LIN {X 0,Y 469.098,Z 495.476,A -85,B 0,C 180,E1 -7636.682,E2 -7636.682} C_VEL
LIN {X 0,Y 468.654,Z 505.589,A -85,B 0,C 180,E1 -7637.503,E2 -7637.503} C_VEL
LIN {X 0,Y 468.178,Z 515.821,A -85,B 0,C 180,E1 -7638.527,E2 -7638.527} C_VEL
LIN {X 0,Y 467.646,Z 524.67,A -85,B 0,C 180,E1 -7639.61,E2 -7639.61} C_VEL
LIN {X 0,Y 467.275,Z 533.304,A -85,B 0,C 180,E1 -7640.913,E2 -7640.913} C_VEL
LIN {X 0,Y 467.012,Z 540.205,A -85,B 0,C 180,E1 -7642.216,E2 -7642.216} C_VEL
LIN {X 0,Y 466.802,Z 545.87,A -85,B 0,C 180,E1 -7643.552,E2 -7643.552} C_VEL
LIN {X 0,Y 466.743,Z 550.076,A -85,B 0,C 180,E1 -7644.816,E2 -7644.816} C_VEL
LIN {X 0,Y 466.652,Z 552.371,A -85,B 0,C 180,E1 -7645.681,E2 -7645.681} C_VEL
LIN {X 0,Y 466.691,Z 554.235,A -85,B 0,C 180,E1 -7646.546,E2 -7646.546} C_VEL
LIN {X 0,Y 466.662,Z 555.631,A -85,B 0,C 180,E1 -7647.41,E2 -7647.41} C_VEL
LIN {X 0,Y 466.618,Z 557.235,A -85,B 0,C 180,E1 -7649.137,E2 -7649.137} C_VEL
LIN {X 0,Y 466.598,Z 557.451,A -85,B 0,C 180,E1 -7650,E2 -7650} C_VEL
LIN {X 0,Y 466.618,Z 557.235,A -85,B 0,C 180,E1 -7650.863,E2 -7650.863} C_VEL
LIN {X 0,Y 466.662,Z 555.634,A -85,B 0,C 180,E1 -7652.589,E2 -7652.589} C_VEL
LIN {X 0,Y 466.691,Z 554.239,A -85,B 0,C 180,E1 -7653.453,E2 -7653.453} C_VEL
LIN {X 0,Y 466.694,Z 551.302,A -85,B 0,C 180,E1 -7654.751,E2 -7654.751} C_VEL
LIN {X 0,Y 466.778,Z 547.328,A -85,B 0,C 180,E1 -7656.05,E2 -7656.05} C_VEL
LIN {X 0,Y 466.979,Z 541.219,A -85,B 0,C 180,E1 -7657.567,E2 -7657.567} C_VEL
LIN {X 0,Y 467.24,Z 534.542,A -85,B 0,C 180,E1 -7658.869,E2 -7658.869} C_VEL
LIN {X 0,Y 467.587,Z 526.257,A -85,B 0,C 180,E1 -7660.172,E2 -7660.172} C_VEL
LIN {X 0,Y 468.054,Z 517.77,A -85,B 0,C 180,E1 -7661.256,E2 -7661.256} C_VEL
LIN {X 0,Y 468.531,Z 507.664,A -85,B 0,C 180,E1 -7662.306,E2 -7662.306} C_VEL
LIN {X 0,Y 469.029,Z 495.903,A -85,B 0,C 180,E1 -7663.286,E2 -7663.286} C_VEL
LIN {X 0,Y 469.583,Z 483.606,A -85,B 0,C 180,E1 -7664.076,E2 -7664.076} C_VEL
LIN {X 0,Y 470.068,Z 471.26,A -85,B 0,C 180,E1 -7664.669,E2 -7664.669} C_VEL
LIN {X 0,Y 468.242,Z 458.397,A -85,B 0,C 180,E1 -7665.176,E2 -7665.176} C_VEL
LIN {X 0,Y 466.978,Z 450.681,A -85,B 0,C 180,E1 -7665.416,E2 -7665.416} C_VEL
LIN {X 0,Y 467.142,Z 442.978,A -85,B 0,C 180,E1 -7668.591,E2 -7668.591} C_VEL
LIN {X 0,Y 467.356,Z 435.681,A -85,B 0,C 180,E1 -7671.618,E2 -7671.618} C_VEL
LIN {X 0,Y 467.577,Z 427.867,A -85,B 0,C 180,E1 -7674.889,E2 -7674.889} C_VEL
LIN {X 0,Y 467.867,Z 420.073,A -85,B 0,C 180,E1 -7678.24,E2 -7678.24} C_VEL
LIN {X 0,Y 468.152,Z 413.506,A -85,B 0,C 180,E1 -7681.163,E2 -7681.163} C_VEL
LIN {X 0,Y 468.441,Z 407.928,A -85,B 0,C 180,E1 -7683.718,E2 -7683.718} C_VEL
LIN {X 0,Y 468.502,Z 403.343,A -85,B 0,C 180,E1 -7685.899,E2 -7685.899} C_VEL
LIN {X 0,Y 467.759,Z 397.999,A -85,B 0,C 180,E1 -7688.621,E2 -7688.621} C_VEL
LIN {X 0,Y 467.622,Z 397.24,A -85,B 0,C 180,E1 -7689.141,E2 -7689.141} C_VEL
LIN {X 0,Y 467.588,Z 397.241,A -85,B 0,C 180,E1 -7692.567,E2 -7692.567} C_VEL
LIN {X 0,Y 467.572,Z 397.243,A -85,B 0,C 180,E1 -7695.053,E2 -7695.053} C_VEL
LIN {X 0,Y 467.59,Z 397.24,A -85,B 0,C 180,E1 -7697.44,E2 -7697.44} C_VEL
LIN {X 0,Y 467.584,Z 397.243,A -85,B 0,C 180,E1 -7700.855,E2 -7700.855} C_VEL
LIN {X 0,Y 467.564,Z 397.244,A -85,B 0,C 180,E1 -7704.26,E2 -7704.26} C_VEL
LIN {X 0,Y 467.583,Z 397.243,A -85,B 0,C 180,E1 -7707.321,E2 -7707.321} C_VEL
LIN {X 0,Y 467.572,Z 397.244,A -85,B 0,C 180,E1 -7710.667,E2 -7710.667} C_VEL
LIN {X 0,Y 467.614,Z 397.236,A -85,B 0,C 180,E1 -7713.199,E2 -7713.199} C_VEL
LIN {X 0,Y 467.592,Z 397.241,A -85,B 0,C 180,E1 -7716.469,E2 -7716.469} C_VEL
LIN {X 0,Y 467.626,Z 397.236,A -85,B 0,C 180,E1 -7719.777,E2 -7719.777} C_VEL
LIN {X 0,Y 467.611,Z 397.239,A -85,B 0,C 180,E1 -7722.507,E2 -7722.507} C_VEL
LIN {X 0,Y 467.608,Z 397.235,A -85,B 0,C 180,E1 -7725.197,E2 -7725.197} C_VEL
LIN {X 0,Y 467.685,Z 397.228,A -85,B 0,C 180,E1 -7727.855,E2 -7727.855} C_VEL
LIN {X 0,Y 467.684,Z 397.228,A -85,B 0,C 180,E1 -7731.357,E2 -7731.357} C_VEL
LIN {X 0,Y 467.745,Z 397.22,A -85,B 0,C 180,E1 -7733.963,E2 -7733.963} C_VEL
LIN {X 0,Y 467.861,Z 397.204,A -85,B 0,C 180,E1 -7737.417,E2 -7737.417} C_VEL
LIN {X 0,Y 467.885,Z 397.206,A -85,B 0,C 180,E1 -7740,E2 -7740} C_VEL
LIN {X 0,Y 467.86,Z 397.206,A -85,B 0,C 180,E1 -7742.583,E2 -7742.583} C_VEL
LIN {X 0,Y 467.746,Z 397.221,A -85,B 0,C 180,E1 -7746.037,E2 -7746.037} C_VEL
LIN {X 0,Y 467.684,Z 397.229,A -85,B 0,C 180,E1 -7748.643,E2 -7748.643} C_VEL
LIN {X 0,Y 467.685,Z 397.23,A -85,B 0,C 180,E1 -7752.145,E2 -7752.145} C_VEL
LIN {X 0,Y 467.651,Z 397.233,A -85,B 0,C 180,E1 -7755.885,E2 -7755.885} C_VEL
LIN {X 0,Y 467.625,Z 397.237,A -85,B 0,C 180,E1 -7759.308,E2 -7759.308} C_VEL
LIN {X 0,Y 467.536,Z 397.25,A -85,B 0,C 180,E1 -7762.074,E2 -7762.074} C_VEL
LIN {X 0,Y 467.587,Z 397.238,A -85,B 0,C 180,E1 -7764.888,E2 -7764.888} C_VEL
LIN {X 0,Y 467.629,Z 397.236,A -85,B 0,C 180,E1 -7767.769,E2 -7767.769} C_VEL
LIN {X 0,Y 467.57,Z 397.244,A -85,B 0,C 180,E1 -7771.045,E2 -7771.045} C_VEL
LIN {X 0,Y 467.592,Z 397.24,A -85,B 0,C 180,E1 -7774.243,E2 -7774.243} C_VEL
LIN {X 0,Y 467.553,Z 397.244,A -85,B 0,C 180,E1 -7777.187,E2 -7777.187} C_VEL
LIN {X 0,Y 467.58,Z 397.239,A -85,B 0,C 180,E1 -7780.265,E2 -7780.265} C_VEL
LIN {X 0,Y 467.588,Z 397.239,A -85,B 0,C 180,E1 -7782.567,E2 -7782.567} C_VEL
LIN {X 0,Y 467.573,Z 397.244,A -85,B 0,C 180,E1 -7785.053,E2 -7785.053} C_VEL
LIN {X 0,Y 467.591,Z 397.241,A -85,B 0,C 180,E1 -7787.44,E2 -7787.44} C_VEL
LIN {X 0,Y 467.584,Z 397.24,A -85,B 0,C 180,E1 -7790.855,E2 -7790.855} C_VEL
LIN {X 0,Y 467.475,Z 397.255,A -85,B 0,C 180,E1 -7794.103,E2 -7794.103} C_VEL
LIN {X 0,Y 467.429,Z 397.919,A -85,B 0,C 180,E1 -7795.156,E2 -7795.156} C_VEL
LIN {X 0,Y 467.372,Z 402.107,A -85,B 0,C 180,E1 -7798.244,E2 -7798.244} C_VEL
LIN {X 0,Y 467.244,Z 406.279,A -85,B 0,C 180,E1 -7801.228,E2 -7801.228} C_VEL
LIN {X 0,Y 467.14,Z 410.962,A -85,B 0,C 180,E1 -7804.514,E2 -7804.514} C_VEL
LIN {X 0,Y 467.04,Z 414.543,A -85,B 0,C 180,E1 -7806.968,E2 -7806.968} C_VEL
LIN {X 0,Y 466.898,Z 418.715,A -85,B 0,C 180,E1 -7809.744,E2 -7809.744} C_VEL
LIN {X 0,Y 466.851,Z 422.911,A -85,B 0,C 180,E1 -7812.478,E2 -7812.478} C_VEL
LIN {X 0,Y 466.817,Z 424.912,A -85,B 0,C 180,E1 -7813.735,E2 -7813.735} C_VEL
LIN {X 0,Y 466.734,Z 426.081,A -85,B 0,C 180,E1 -7814.067,E2 -7814.067} C_VEL
LIN {X 0,Y 466.42,Z 428.863,A -85,B 0,C 180,E1 -7814.419,E2 -7814.419} C_VEL
LIN {X 0,Y 465.81,Z 433.444,A -85,B 0,C 180,E1 -7814.735,E2 -7814.735} C_VEL
LIN {X 0,Y 465.219,Z 437.43,A -85,B 0,C 180,E1 -7814.919,E2 -7814.919} C_VEL
LIN {X 0,Y 463.985,Z 445.772,A -85,B 0,C 180,E1 -7815.2,E2 -7815.2} C_VEL
LIN {X 0,Y 463.149,Z 452.928,A -85,B 0,C 180,E1 -7815.511,E2 -7815.511} C_VEL
LIN {X 0,Y 462.676,Z 464.1,A -85,B 0,C 180,E1 -7816.159,E2 -7816.159} C_VEL
LIN {X 0,Y 462.246,Z 474.476,A -85,B 0,C 180,E1 -7816.929,E2 -7816.929} C_VEL
LIN {X 0,Y 461.72,Z 485.163,A -85,B 0,C 180,E1 -7817.919,E2 -7817.919} C_VEL
LIN {X 0,Y 461.147,Z 494.78,A -85,B 0,C 180,E1 -7819.018,E2 -7819.018} C_VEL
LIN {X 0,Y 460.748,Z 502.654,A -85,B 0,C 180,E1 -7820.119,E2 -7820.119} C_VEL
LIN {X 0,Y 460.319,Z 510.353,A -85,B 0,C 180,E1 -7821.439,E2 -7821.439} C_VEL
LIN {X 0,Y 459.943,Z 517.415,A -85,B 0,C 180,E1 -7822.979,E2 -7822.979} C_VEL
LIN {X 0,Y 459.872,Z 522.116,A -85,B 0,C 180,E1 -7824.299,E2 -7824.299} C_VEL
LIN {X 0,Y 459.676,Z 525.72,A -85,B 0,C 180,E1 -7825.616,E2 -7825.616} C_VEL
LIN {X 0,Y 459.707,Z 527.58,A -85,B 0,C 180,E1 -7826.494,E2 -7826.494} C_VEL
LIN {X 0,Y 459.608,Z 528.985,A -85,B 0,C 180,E1 -7827.371,E2 -7827.371} C_VEL
LIN {X 0,Y 459.523,Z 530.598,A -85,B 0,C 180,E1 -7829.124,E2 -7829.124} C_VEL
LIN {X 0,Y 459.53,Z 530.833,A -85,B 0,C 180,E1 -7830,E2 -7830} C_VEL
LIN {X 0,Y 459.523,Z 530.646,A -85,B 0,C 180,E1 -7830.876,E2 -7830.876} C_VEL
LIN {X 0,Y 459.608,Z 529.096,A -85,B 0,C 180,E1 -7832.629,E2 -7832.629} C_VEL
LIN {X 0,Y 459.689,Z 527.741,A -85,B 0,C 180,E1 -7833.506,E2 -7833.506} C_VEL
LIN {X 0,Y 459.671,Z 524.88,A -85,B 0,C 180,E1 -7834.824,E2 -7834.824} C_VEL
LIN {X 0,Y 459.921,Z 520.994,A -85,B 0,C 180,E1 -7836.141,E2 -7836.141} C_VEL
LIN {X 0,Y 460.047,Z 515.986,A -85,B 0,C 180,E1 -7837.461,E2 -7837.461} C_VEL
LIN {X 0,Y 460.375,Z 509.678,A -85,B 0,C 180,E1 -7838.781,E2 -7838.781} C_VEL
LIN {X 0,Y 460.73,Z 501.782,A -85,B 0,C 180,E1 -7840.103,E2 -7840.103} C_VEL
LIN {X 0,Y 461.286,Z 491.956,A -85,B 0,C 180,E1 -7841.424,E2 -7841.424} C_VEL
LIN {X 0,Y 461.937,Z 481.725,A -85,B 0,C 180,E1 -7842.514,E2 -7842.514} C_VEL
LIN {X 0,Y 462.338,Z 470.839,A -85,B 0,C 180,E1 -7843.451,E2 -7843.451} C_VEL
LIN {X 0,Y 462.833,Z 460.258,A -85,B 0,C 180,E1 -7844.173,E2 -7844.173} C_VEL
LIN {X 0,Y 463.274,Z 447.688,A -85,B 0,C 180,E1 -7844.833,E2 -7844.833} C_VEL
LIN {X 0,Y 463.206,Z 443.667,A -85,B 0,C 180,E1 -7845.01,E2 -7845.01} C_VEL
LIN {X 0,Y 460.798,Z 431.07,A -85,B 0,C 180,E1 -7845.515,E2 -7845.515} C_VEL
LIN {X 0,Y 459.769,Z 426.584,A -85,B 0,C 180,E1 -7845.672,E2 -7845.672} C_VEL
LIN {X 0,Y 459.841,Z 421.829,A -85,B 0,C 180,E1 -7848.721,E2 -7848.721} C_VEL
LIN {X 0,Y 459.92,Z 416.213,A -85,B 0,C 180,E1 -7852.459,E2 -7852.459} C_VEL
LIN {X 0,Y 460.066,Z 411.592,A -85,B 0,C 180,E1 -7855.672,E2 -7855.672} C_VEL
LIN {X 0,Y 460.258,Z 406.541,A -85,B 0,C 180,E1 -7859.251,E2 -7859.251} C_VEL
LIN {X 0,Y 460.328,Z 402.349,A -85,B 0,C 180,E1 -7862.301,E2 -7862.301} C_VEL
LIN {X 0,Y 460.414,Z 399.416,A -85,B 0,C 180,E1 -7864.484,E2 -7864.484} C_VEL
LIN {X 0,Y 460.367,Z 398.143,A -85,B 0,C 180,E1 -7865.459,E2 -7865.459} C_VEL
LIN {X 0,Y 460.499,Z 398.121,A -85,B 0,C 180,E1 -7867.624,E2 -7867.624} C_VEL
LIN {X 0,Y 460.546,Z 398.118,A -85,B 0,C 180,E1 -7870.27,E2 -7870.27} C_VEL
LIN {X 0,Y 460.511,Z 398.123,A -85,B 0,C 180,E1 -7873.374,E2 -7873.374} C_VEL
LIN {X 0,Y 460.499,Z 398.124,A -85,B 0,C 180,E1 -7876.624,E2 -7876.624} C_VEL
LIN {X 0,Y 460.545,Z 398.115,A -85,B 0,C 180,E1 -7879.731,E2 -7879.731} C_VEL
LIN {X 0,Y 460.529,Z 398.122,A -85,B 0,C 180,E1 -7882.52,E2 -7882.52} C_VEL
LIN {X 0,Y 460.549,Z 398.117,A -85,B 0,C 180,E1 -7885.624,E2 -7885.624} C_VEL
LIN {X 0,Y 460.54,Z 398.12,A -85,B 0,C 180,E1 -7888.745,E2 -7888.745} C_VEL
LIN {X 0,Y 460.592,Z 398.113,A -85,B 0,C 180,E1 -7892.252,E2 -7892.252} C_VEL
LIN {X 0,Y 460.534,Z 398.117,A -85,B 0,C 180,E1 -7895.667,E2 -7895.667} C_VEL
LIN {X 0,Y 460.524,Z 398.12,A -85,B 0,C 180,E1 -7898.578,E2 -7898.578} C_VEL
LIN {X 0,Y 460.59,Z 398.112,A -85,B 0,C 180,E1 -7901.311,E2 -7901.311} C_VEL
LIN {X 0,Y 460.607,Z 398.11,A -85,B 0,C 180,E1 -7904.059,E2 -7904.059} C_VEL
LIN {X 0,Y 460.613,Z 398.108,A -85,B 0,C 180,E1 -7907.666,E2 -7907.666} C_VEL
LIN {X 0,Y 460.632,Z 398.106,A -85,B 0,C 180,E1 -7911.224,E2 -7911.224} C_VEL
LIN {X 0,Y 460.713,Z 398.097,A -85,B 0,C 180,E1 -7913.87,E2 -7913.87} C_VEL
LIN {X 0,Y 460.802,Z 398.085,A -85,B 0,C 180,E1 -7917.377,E2 -7917.377} C_VEL
LIN {X 0,Y 460.856,Z 398.082,A -85,B 0,C 180,E1 -7920,E2 -7920} C_VEL
LIN {X 0,Y 460.803,Z 398.083,A -85,B 0,C 180,E1 -7922.622,E2 -7922.622} C_VEL
LIN {X 0,Y 460.713,Z 398.097,A -85,B 0,C 180,E1 -7926.13,E2 -7926.13} C_VEL
LIN {X 0,Y 460.632,Z 398.107,A -85,B 0,C 180,E1 -7928.776,E2 -7928.776} C_VEL
LIN {X 0,Y 460.638,Z 398.105,A -85,B 0,C 180,E1 -7932.457,E2 -7932.457} C_VEL
LIN {X 0,Y 460.603,Z 398.109,A -85,B 0,C 180,E1 -7935.997,E2 -7935.997} C_VEL
LIN {X 0,Y 460.575,Z 398.115,A -85,B 0,C 180,E1 -7938.902,E2 -7938.902} C_VEL
LIN {X 0,Y 460.519,Z 398.121,A -85,B 0,C 180,E1 -7941.486,E2 -7941.486} C_VEL
LIN {X 0,Y 460.534,Z 398.118,A -85,B 0,C 180,E1 -7944.333,E2 -7944.333} C_VEL
LIN {X 0,Y 460.591,Z 398.111,A -85,B 0,C 180,E1 -7947.748,E2 -7947.748} C_VEL
LIN {X 0,Y 460.523,Z 398.121,A -85,B 0,C 180,E1 -7951.283,E2 -7951.283} C_VEL
LIN {X 0,Y 460.536,Z 398.12,A -85,B 0,C 180,E1 -7954.506,E2 -7954.506} C_VEL
LIN {X 0,Y 460.531,Z 398.12,A -85,B 0,C 180,E1 -7957.62,E2 -7957.62} C_VEL
LIN {X 0,Y 460.544,Z 398.116,A -85,B 0,C 180,E1 -7960.269,E2 -7960.269} C_VEL
LIN {X 0,Y 460.503,Z 398.122,A -85,B 0,C 180,E1 -7963.375,E2 -7963.375} C_VEL
LIN {X 0,Y 460.512,Z 398.124,A -85,B 0,C 180,E1 -7966.626,E2 -7966.626} C_VEL
LIN {X 0,Y 460.545,Z 398.123,A -85,B 0,C 180,E1 -7969.73,E2 -7969.73} C_VEL
LIN {X 0,Y 460.596,Z 398.172,A -85,B 0,C 180,E1 -7970.781,E2 -7970.781} C_VEL
LIN {X 0,Y 461.478,Z 403.993,A -85,B 0,C 180,E1 -7973.819,E2 -7973.819} C_VEL
LIN {X 0,Y 461.428,Z 408.951,A -85,B 0,C 180,E1 -7976.225,E2 -7976.225} C_VEL
LIN {X 0,Y 461.086,Z 416.657,A -85,B 0,C 180,E1 -7979.801,E2 -7979.801} C_VEL
LIN {X 0,Y 460.697,Z 423.307,A -85,B 0,C 180,E1 -7982.764,E2 -7982.764} C_VEL
LIN {X 0,Y 460.487,Z 429.977,A -85,B 0,C 180,E1 -7985.664,E2 -7985.664} C_VEL
LIN {X 0,Y 460.278,Z 436.992,A -85,B 0,C 180,E1 -7988.656,E2 -7988.656} C_VEL
LIN {X 0,Y 460.04,Z 444.334,A -85,B 0,C 180,E1 -7991.749,E2 -7991.749} C_VEL
LIN {X 0,Y 459.912,Z 450.511,A -85,B 0,C 180,E1 -7994.351,E2 -7994.351} C_VEL
LIN {X 0,Y 462.129,Z 464.356,A -85,B 0,C 180,E1 -7994.812,E2 -7994.812} C_VEL
LIN {X 0,Y 463.103,Z 472.383,A -85,B 0,C 180,E1 -7995.162,E2 -7995.162} C_VEL
LIN {X 0,Y 462.697,Z 483.416,A -85,B 0,C 180,E1 -7995.71,E2 -7995.71} C_VEL
LIN {X 0,Y 462.168,Z 495.274,A -85,B 0,C 180,E1 -7996.479,E2 -7996.479} C_VEL
LIN {X 0,Y 461.66,Z 505.773,A -85,B 0,C 180,E1 -7997.347,E2 -7997.347} C_VEL
LIN {X 0,Y 461.19,Z 515.618,A -85,B 0,C 180,E1 -7998.351,E2 -7998.351} C_VEL
LIN {X 0,Y 460.632,Z 524.467,A -85,B 0,C 180,E1 -7999.45,E2 -7999.45} C_VEL
LIN {X 0,Y 460.241,Z 533.1,A -85,B 0,C 180,E1 -8000.773,E2 -8000.773} C_VEL
LIN {X 0,Y 459.951,Z 540.001,A -85,B 0,C 180,E1 -8002.096,E2 -8002.096} C_VEL
LIN {X 0,Y 459.713,Z 546.099,A -85,B 0,C 180,E1 -8003.57,E2 -8003.57} C_VEL
LIN {X 0,Y 459.622,Z 551.097,A -85,B 0,C 180,E1 -8005.176,E2 -8005.176} C_VEL
LIN {X 0,Y 459.586,Z 554.031,A -85,B 0,C 180,E1 -8006.493,E2 -8006.493} C_VEL
LIN {X 0,Y 459.584,Z 555.428,A -85,B 0,C 180,E1 -8007.37,E2 -8007.37} C_VEL
LIN {X 0,Y 459.521,Z 557.031,A -85,B 0,C 180,E1 -8009.124,E2 -8009.124} C_VEL
LIN {X 0,Y 459.53,Z 557.248,A -85,B 0,C 180,E1 -8010,E2 -8010} C_VEL
LIN {X 0,Y 459.521,Z 557.031,A -85,B 0,C 180,E1 -8010.876,E2 -8010.876} C_VEL
LIN {X 0,Y 459.584,Z 555.43,A -85,B 0,C 180,E1 -8012.629,E2 -8012.629} C_VEL
LIN {X 0,Y 459.586,Z 554.034,A -85,B 0,C 180,E1 -8013.507,E2 -8013.507} C_VEL
LIN {X 0,Y 459.622,Z 551.098,A -85,B 0,C 180,E1 -8014.824,E2 -8014.824} C_VEL
LIN {X 0,Y 459.713,Z 546.096,A -85,B 0,C 180,E1 -8016.43,E2 -8016.43} C_VEL
LIN {X 0,Y 459.951,Z 540,A -85,B 0,C 180,E1 -8017.904,E2 -8017.904} C_VEL
LIN {X 0,Y 460.241,Z 533.098,A -85,B 0,C 180,E1 -8019.226,E2 -8019.226} C_VEL
LIN {X 0,Y 460.632,Z 524.463,A -85,B 0,C 180,E1 -8020.55,E2 -8020.55} C_VEL
LIN {X 0,Y 461.186,Z 515.612,A -85,B 0,C 180,E1 -8021.649,E2 -8021.649} C_VEL
LIN {X 0,Y 461.707,Z 505.837,A -85,B 0,C 180,E1 -8022.645,E2 -8022.645} C_VEL
LIN {X 0,Y 462.142,Z 495.266,A -85,B 0,C 180,E1 -8023.522,E2 -8023.522} C_VEL
LIN {X 0,Y 462.684,Z 483.397,A -85,B 0,C 180,E1 -8024.29,E2 -8024.29} C_VEL
LIN {X 0,Y 463.112,Z 471.048,A -85,B 0,C 180,E1 -8024.894,E2 -8024.894} C_VEL
LIN {X 0,Y 461.147,Z 457.996,A -85,B 0,C 180,E1 -8025.421,E2 -8025.421} C_VEL
LIN {X 0,Y 459.913,Z 450.507,A -85,B 0,C 180,E1 -8025.649,E2 -8025.649} C_VEL
LIN {X 0,Y 460.102,Z 442.235,A -85,B 0,C 180,E1 -8029.126,E2 -8029.126} C_VEL
LIN {X 0,Y 460.306,Z 435.521,A -85,B 0,C 180,E1 -8031.967,E2 -8031.967} C_VEL
LIN {X 0,Y 460.573,Z 427.726,A -85,B 0,C 180,E1 -8035.294,E2 -8035.294} C_VEL
LIN {X 0,Y 460.903,Z 419.951,A -85,B 0,C 180,E1 -8038.706,E2 -8038.706} C_VEL
LIN {X 0,Y 461.171,Z 413.989,A -85,B 0,C 180,E1 -8041.415,E2 -8041.415} C_VEL
LIN {X 0,Y 461.515,Z 407.028,A -85,B 0,C 180,E1 -8044.682,E2 -8044.682} C_VEL
LIN {X 0,Y 461.253,Z 402.369,A -85,B 0,C 180,E1 -8047.003,E2 -8047.003} C_VEL
LIN {X 0,Y 460.56,Z 398.119,A -85,B 0,C 180,E1 -8049.348,E2 -8049.348} C_VEL
LIN {X 0,Y 460.525,Z 398.124,A -85,B 0,C 180,E1 -8052.181,E2 -8052.181} C_VEL
LIN {X 0,Y 460.519,Z 398.124,A -85,B 0,C 180,E1 -8055.411,E2 -8055.411} C_VEL
LIN {X 0,Y 460.533,Z 398.117,A -85,B 0,C 180,E1 -8058.397,E2 -8058.397} C_VEL
LIN {X 0,Y 460.528,Z 398.119,A -85,B 0,C 180,E1 -8061.267,E2 -8061.267} C_VEL
LIN {X 0,Y 460.515,Z 398.123,A -85,B 0,C 180,E1 -8064.555,E2 -8064.555} C_VEL
LIN {X 0,Y 460.533,Z 398.118,A -85,B 0,C 180,E1 -8067.716,E2 -8067.716} C_VEL
LIN {X 0,Y 460.542,Z 398.121,A -85,B 0,C 180,E1 -8070.769,E2 -8070.769} C_VEL
LIN {X 0,Y 460.557,Z 398.114,A -85,B 0,C 180,E1 -8073.734,E2 -8073.734} C_VEL
LIN {X 0,Y 460.546,Z 398.118,A -85,B 0,C 180,E1 -8076.624,E2 -8076.624} C_VEL
LIN {X 0,Y 460.554,Z 398.116,A -85,B 0,C 180,E1 -8079.453,E2 -8079.453} C_VEL
LIN {X 0,Y 460.561,Z 398.115,A -85,B 0,C 180,E1 -8082.23,E2 -8082.23} C_VEL
LIN {X 0,Y 460.567,Z 398.114,A -85,B 0,C 180,E1 -8084.965,E2 -8084.965} C_VEL
LIN {X 0,Y 460.632,Z 398.106,A -85,B 0,C 180,E1 -8087.666,E2 -8087.666} C_VEL
LIN {X 0,Y 460.631,Z 398.107,A -85,B 0,C 180,E1 -8091.224,E2 -8091.224} C_VEL
LIN {X 0,Y 460.712,Z 398.097,A -85,B 0,C 180,E1 -8093.87,E2 -8093.87} C_VEL
LIN {X 0,Y 460.802,Z 398.083,A -85,B 0,C 180,E1 -8097.378,E2 -8097.378} C_VEL
LIN {X 0,Y 460.856,Z 398.081,A -85,B 0,C 180,E1 -8100,E2 -8100} C_VEL
LIN {X 0,Y 460.801,Z 398.085,A -85,B 0,C 180,E1 -8102.623,E2 -8102.623} C_VEL
LIN {X 0,Y 460.712,Z 398.097,A -85,B 0,C 180,E1 -8106.13,E2 -8106.13} C_VEL
LIN {X 0,Y 460.631,Z 398.106,A -85,B 0,C 180,E1 -8108.776,E2 -8108.776} C_VEL
LIN {X 0,Y 460.636,Z 398.105,A -85,B 0,C 180,E1 -8112.457,E2 -8112.457} C_VEL
LIN {X 0,Y 460.602,Z 398.111,A -85,B 0,C 180,E1 -8115.998,E2 -8115.998} C_VEL
LIN {X 0,Y 460.571,Z 398.115,A -85,B 0,C 180,E1 -8119.616,E2 -8119.616} C_VEL
LIN {X 0,Y 460.513,Z 398.121,A -85,B 0,C 180,E1 -8122.429,E2 -8122.429} C_VEL
LIN {X 0,Y 460.555,Z 398.119,A -85,B 0,C 180,E1 -8125.798,E2 -8125.798} C_VEL
LIN {X 0,Y 460.557,Z 398.115,A -85,B 0,C 180,E1 -8128.233,E2 -8128.233} C_VEL
LIN {X 0,Y 460.523,Z 398.122,A -85,B 0,C 180,E1 -8131.283,E2 -8131.283} C_VEL
LIN {X 0,Y 460.536,Z 398.118,A -85,B 0,C 180,E1 -8134.506,E2 -8134.506} C_VEL
LIN {X 0,Y 460.531,Z 398.123,A -85,B 0,C 180,E1 -8137.621,E2 -8137.621} C_VEL
LIN {X 0,Y 460.544,Z 398.115,A -85,B 0,C 180,E1 -8140.27,E2 -8140.27} C_VEL
LIN {X 0,Y 460.502,Z 398.124,A -85,B 0,C 180,E1 -8143.375,E2 -8143.375} C_VEL
LIN {X 0,Y 460.511,Z 398.122,A -85,B 0,C 180,E1 -8146.626,E2 -8146.626} C_VEL
LIN {X 0,Y 460.545,Z 398.118,A -85,B 0,C 180,E1 -8149.731,E2 -8149.731} C_VEL
LIN {X 0,Y 460.495,Z 398.121,A -85,B 0,C 180,E1 -8152.525,E2 -8152.525} C_VEL
LIN {X 0,Y 460.375,Z 398.142,A -85,B 0,C 180,E1 -8154.542,E2 -8154.542} C_VEL
LIN {X 0,Y 460.355,Z 401.412,A -85,B 0,C 180,E1 -8157.104,E2 -8157.104} C_VEL
LIN {X 0,Y 460.26,Z 405.006,A -85,B 0,C 180,E1 -8159.742,E2 -8159.742} C_VEL
LIN {X 0,Y 460.113,Z 409.176,A -85,B 0,C 180,E1 -8162.727,E2 -8162.727} C_VEL
LIN {X 0,Y 460.003,Z 413.321,A -85,B 0,C 180,E1 -8165.637,E2 -8165.637} C_VEL
LIN {X 0,Y 459.851,Z 417.941,A -85,B 0,C 180,E1 -8168.793,E2 -8168.793} C_VEL
LIN {X 0,Y 459.844,Z 421.815,A -85,B 0,C 180,E1 -8171.366,E2 -8171.366} C_VEL
LIN {X 0,Y 459.814,Z 426.595,A -85,B 0,C 180,E1 -8174.429,E2 -8174.429} C_VEL
LIN {X 0,Y 462.668,Z 440.317,A -85,B 0,C 180,E1 -8174.936,E2 -8174.936} C_VEL
LIN {X 0,Y 463.317,Z 445.574,A -85,B 0,C 180,E1 -8175.169,E2 -8175.169} C_VEL
LIN {X 0,Y 463.149,Z 452.928,A -85,B 0,C 180,E1 -8175.511,E2 -8175.511} C_VEL
LIN {X 0,Y 462.255,Z 458.367,A -85,B 0,C 180,E1 -8175.777,E2 -8175.777} C_VEL
LIN {X 0,Y 459.141,Z 467.025,A -85,B 0,C 180,E1 -8176.238,E2 -8176.238} C_VEL
LIN {X 0,Y 456.005,Z 475.282,A -85,B 0,C 180,E1 -8176.795,E2 -8176.795} C_VEL
LIN {X 0,Y 455.08,Z 480.086,A -85,B 0,C 180,E1 -8177.208,E2 -8177.208} C_VEL
LIN {X 0,Y 454.511,Z 489.458,A -85,B 0,C 180,E1 -8178.177,E2 -8178.177} C_VEL
LIN {X 0,Y 454.035,Z 498.302,A -85,B 0,C 180,E1 -8179.295,E2 -8179.295} C_VEL
LIN {X 0,Y 453.531,Z 506.932,A -85,B 0,C 180,E1 -8180.636,E2 -8180.636} C_VEL
LIN {X 0,Y 453.095,Z 513.811,A -85,B 0,C 180,E1 -8181.975,E2 -8181.975} C_VEL
LIN {X 0,Y 452.869,Z 519.329,A -85,B 0,C 180,E1 -8183.32,E2 -8183.32} C_VEL
LIN {X 0,Y 452.695,Z 523.638,A -85,B 0,C 180,E1 -8184.655,E2 -8184.655} C_VEL
LIN {X 0,Y 452.585,Z 525.926,A -85,B 0,C 180,E1 -8185.547,E2 -8185.547} C_VEL
LIN {X 0,Y 452.622,Z 527.785,A -85,B 0,C 180,E1 -8186.439,E2 -8186.439} C_VEL
LIN {X 0,Y 452.535,Z 529.189,A -85,B 0,C 180,E1 -8187.33,E2 -8187.33} C_VEL
LIN {X 0,Y 452.43,Z 530.802,A -85,B 0,C 180,E1 -8189.11,E2 -8189.11} C_VEL
LIN {X 0,Y 452.435,Z 531.037,A -85,B 0,C 180,E1 -8190,E2 -8190} C_VEL
LIN {X 0,Y 452.43,Z 530.85,A -85,B 0,C 180,E1 -8190.89,E2 -8190.89} C_VEL
LIN {X 0,Y 452.534,Z 529.299,A -85,B 0,C 180,E1 -8192.671,E2 -8192.671} C_VEL
LIN {X 0,Y 452.606,Z 527.944,A -85,B 0,C 180,E1 -8193.561,E2 -8193.561} C_VEL
LIN {X 0,Y 452.603,Z 525.083,A -85,B 0,C 180,E1 -8194.899,E2 -8194.899} C_VEL
LIN {X 0,Y 452.85,Z 521.197,A -85,B 0,C 180,E1 -8196.237,E2 -8196.237} C_VEL
LIN {X 0,Y 452.99,Z 516.188,A -85,B 0,C 180,E1 -8197.578,E2 -8197.578} C_VEL
LIN {X 0,Y 453.357,Z 509.88,A -85,B 0,C 180,E1 -8198.918,E2 -8198.918} C_VEL
LIN {X 0,Y 453.743,Z 501.983,A -85,B 0,C 180,E1 -8200.261,E2 -8200.261} C_VEL
LIN {X 0,Y 454.336,Z 492.156,A -85,B 0,C 180,E1 -8201.601,E2 -8201.601} C_VEL
LIN {X 0,Y 455.009,Z 482.059,A -85,B 0,C 180,E1 -8202.694,E2 -8202.694} C_VEL
LIN {X 0,Y 455.414,Z 471.637,A -85,B 0,C 180,E1 -8203.611,E2 -8203.611} C_VEL
LIN {X 0,Y 455.968,Z 460.454,A -85,B 0,C 180,E1 -8204.391,E2 -8204.391} C_VEL
LIN {X 0,Y 456.413,Z 447.882,A -85,B 0,C 180,E1 -8205.061,E2 -8205.061} C_VEL
LIN {X 0,Y 456.031,Z 442.556,A -85,B 0,C 180,E1 -8205.304,E2 -8205.304} C_VEL
LIN {X 0,Y 453.255,Z 429.318,A -85,B 0,C 180,E1 -8205.83,E2 -8205.83} C_VEL
LIN {X 0,Y 452.664,Z 426.786,A -85,B 0,C 180,E1 -8205.922,E2 -8205.922} C_VEL
LIN {X 0,Y 452.774,Z 422.006,A -85,B 0,C 180,E1 -8209.024,E2 -8209.024} C_VEL
LIN {X 0,Y 452.816,Z 417.78,A -85,B 0,C 180,E1 -8211.87,E2 -8211.87} C_VEL
LIN {X 0,Y 452.962,Z 413.615,A -85,B 0,C 180,E1 -8214.767,E2 -8214.767} C_VEL
LIN {X 0,Y 453.077,Z 409.294,A -85,B 0,C 180,E1 -8217.85,E2 -8217.85} C_VEL
LIN {X 0,Y 453.247,Z 405.268,A -85,B 0,C 180,E1 -8220.777,E2 -8220.777} C_VEL
LIN {X 0,Y 453.346,Z 401.055,A -85,B 0,C 180,E1 -8223.924,E2 -8223.924} C_VEL
LIN {X 0,Y 453.353,Z 399.651,A -85,B 0,C 180,E1 -8225.001,E2 -8225.001} C_VEL
LIN {X 0,Y 453.4,Z 399.009,A -85,B 0,C 180,E1 -8226.289,E2 -8226.289} C_VEL
LIN {X 0,Y 453.492,Z 398.995,A -85,B 0,C 180,E1 -8229.45,E2 -8229.45} C_VEL
LIN {X 0,Y 453.481,Z 398.997,A -85,B 0,C 180,E1 -8231.935,E2 -8231.935} C_VEL
LIN {X 0,Y 453.486,Z 398.997,A -85,B 0,C 180,E1 -8235.471,E2 -8235.471} C_VEL
LIN {X 0,Y 453.482,Z 398.997,A -85,B 0,C 180,E1 -8238.209,E2 -8238.209} C_VEL
LIN {X 0,Y 453.513,Z 398.995,A -85,B 0,C 180,E1 -8240.791,E2 -8240.791} C_VEL
LIN {X 0,Y 453.457,Z 399,A -85,B 0,C 180,E1 -8243.917,E2 -8243.917} C_VEL
LIN {X 0,Y 453.486,Z 398.997,A -85,B 0,C 180,E1 -8247.151,E2 -8247.151} C_VEL
LIN {X 0,Y 453.478,Z 398.998,A -85,B 0,C 180,E1 -8250.268,E2 -8250.268} C_VEL
LIN {X 0,Y 453.508,Z 398.991,A -85,B 0,C 180,E1 -8253.294,E2 -8253.294} C_VEL
LIN {X 0,Y 453.501,Z 398.998,A -85,B 0,C 180,E1 -8256.239,E2 -8256.239} C_VEL
LIN {X 0,Y 453.486,Z 398.996,A -85,B 0,C 180,E1 -8259.118,E2 -8259.118} C_VEL
LIN {X 0,Y 453.507,Z 398.995,A -85,B 0,C 180,E1 -8261.944,E2 -8261.944} C_VEL
LIN {X 0,Y 453.543,Z 398.99,A -85,B 0,C 180,E1 -8264.726,E2 -8264.726} C_VEL
LIN {X 0,Y 453.563,Z 398.987,A -85,B 0,C 180,E1 -8268.379,E2 -8268.379} C_VEL
LIN {X 0,Y 453.656,Z 398.977,A -85,B 0,C 180,E1 -8271.985,E2 -8271.985} C_VEL
LIN {X 0,Y 453.673,Z 398.974,A -85,B 0,C 180,E1 -8274.667,E2 -8274.667} C_VEL
LIN {X 0,Y 453.746,Z 398.964,A -85,B 0,C 180,E1 -8277.337,E2 -8277.337} C_VEL
LIN {X 0,Y 453.826,Z 398.957,A -85,B 0,C 180,E1 -8280,E2 -8280} C_VEL
LIN {X 0,Y 453.747,Z 398.962,A -85,B 0,C 180,E1 -8282.663,E2 -8282.663} C_VEL
LIN {X 0,Y 453.68,Z 398.973,A -85,B 0,C 180,E1 -8286.225,E2 -8286.225} C_VEL
LIN {X 0,Y 453.596,Z 398.983,A -85,B 0,C 180,E1 -8288.913,E2 -8288.913} C_VEL
LIN {X 0,Y 453.605,Z 398.98,A -85,B 0,C 180,E1 -8292.551,E2 -8292.551} C_VEL
LIN {X 0,Y 453.548,Z 398.987,A -85,B 0,C 180,E1 -8296.196,E2 -8296.196} C_VEL
LIN {X 0,Y 453.524,Z 398.994,A -85,B 0,C 180,E1 -8299.041,E2 -8299.041} C_VEL
LIN {X 0,Y 453.479,Z 399,A -85,B 0,C 180,E1 -8301.836,E2 -8301.836} C_VEL
LIN {X 0,Y 453.504,Z 398.995,A -85,B 0,C 180,E1 -8304.735,E2 -8304.735} C_VEL
LIN {X 0,Y 453.54,Z 398.988,A -85,B 0,C 180,E1 -8307.961,E2 -8307.961} C_VEL
LIN {X 0,Y 453.468,Z 398.999,A -85,B 0,C 180,E1 -8311.525,E2 -8311.525} C_VEL
LIN {X 0,Y 453.491,Z 398.998,A -85,B 0,C 180,E1 -8314.778,E2 -8314.778} C_VEL
LIN {X 0,Y 453.476,Z 398.998,A -85,B 0,C 180,E1 -8318.311,E2 -8318.311} C_VEL
LIN {X 0,Y 453.496,Z 398.995,A -85,B 0,C 180,E1 -8320.609,E2 -8320.609} C_VEL
LIN {X 0,Y 453.459,Z 399,A -85,B 0,C 180,E1 -8323.244,E2 -8323.244} C_VEL
LIN {X 0,Y 453.476,Z 398.998,A -85,B 0,C 180,E1 -8325.78,E2 -8325.78} C_VEL
LIN {X 0,Y 453.484,Z 399.003,A -85,B 0,C 180,E1 -8328.21,E2 -8328.21} C_VEL
LIN {X 0,Y 453.533,Z 399.042,A -85,B 0,C 180,E1 -8330.555,E2 -8330.555} C_VEL
LIN {X 0,Y 454.425,Z 404.644,A -85,B 0,C 180,E1 -8333.535,E2 -8333.535} C_VEL
LIN {X 0,Y 454.472,Z 408.858,A -85,B 0,C 180,E1 -8335.636,E2 -8335.636} C_VEL
LIN {X 0,Y 454.114,Z 415.52,A -85,B 0,C 180,E1 -8338.807,E2 -8338.807} C_VEL
LIN {X 0,Y 453.881,Z 420.959,A -85,B 0,C 180,E1 -8341.314,E2 -8341.314} C_VEL
LIN {X 0,Y 453.507,Z 428.719,A -85,B 0,C 180,E1 -8344.775,E2 -8344.775} C_VEL
LIN {X 0,Y 453.237,Z 436.47,A -85,B 0,C 180,E1 -8348.152,E2 -8348.152} C_VEL
LIN {X 0,Y 453.005,Z 443.441,A -85,B 0,C 180,E1 -8351.15,E2 -8351.15} C_VEL
LIN {X 0,Y 452.869,Z 450.487,A -85,B 0,C 180,E1 -8354.112,E2 -8354.112} C_VEL
LIN {X 0,Y 455.035,Z 463.693,A -85,B 0,C 180,E1 -8354.552,E2 -8354.552} C_VEL
LIN {X 0,Y 456.209,Z 473.487,A -85,B 0,C 180,E1 -8354.989,E2 -8354.989} C_VEL
LIN {X 0,Y 455.72,Z 485.136,A -85,B 0,C 180,E1 -8355.601,E2 -8355.601} C_VEL
LIN {X 0,Y 455.156,Z 496.501,A -85,B 0,C 180,E1 -8356.38,E2 -8356.38} C_VEL
LIN {X 0,Y 454.614,Z 507.617,A -85,B 0,C 180,E1 -8357.345,E2 -8357.345} C_VEL
LIN {X 0,Y 454.082,Z 517.365,A -85,B 0,C 180,E1 -8358.392,E2 -8358.392} C_VEL
LIN {X 0,Y 453.528,Z 525.85,A -85,B 0,C 180,E1 -8359.509,E2 -8359.509} C_VEL
LIN {X 0,Y 453.125,Z 534.133,A -85,B 0,C 180,E1 -8360.852,E2 -8360.852} C_VEL
LIN {X 0,Y 452.842,Z 540.81,A -85,B 0,C 180,E1 -8362.195,E2 -8362.195} C_VEL
LIN {X 0,Y 452.604,Z 546.921,A -85,B 0,C 180,E1 -8363.76,E2 -8363.76} C_VEL
LIN {X 0,Y 452.55,Z 550.894,A -85,B 0,C 180,E1 -8365.1,E2 -8365.1} C_VEL
LIN {X 0,Y 452.483,Z 553.827,A -85,B 0,C 180,E1 -8366.438,E2 -8366.438} C_VEL
LIN {X 0,Y 452.508,Z 555.224,A -85,B 0,C 180,E1 -8367.329,E2 -8367.329} C_VEL
LIN {X 0,Y 452.428,Z 556.827,A -85,B 0,C 180,E1 -8369.11,E2 -8369.11} C_VEL
LIN {X 0,Y 452.434,Z 557.044,A -85,B 0,C 180,E1 -8370,E2 -8370} C_VEL
LIN {X 0,Y 452.428,Z 556.827,A -85,B 0,C 180,E1 -8370.89,E2 -8370.89} C_VEL
LIN {X 0,Y 452.508,Z 555.227,A -85,B 0,C 180,E1 -8372.671,E2 -8372.671} C_VEL
LIN {X 0,Y 452.482,Z 553.829,A -85,B 0,C 180,E1 -8373.562,E2 -8373.562} C_VEL
LIN {X 0,Y 452.55,Z 550.893,A -85,B 0,C 180,E1 -8374.9,E2 -8374.9} C_VEL
LIN {X 0,Y 452.628,Z 546.307,A -85,B 0,C 180,E1 -8376.416,E2 -8376.416} C_VEL
LIN {X 0,Y 452.893,Z 539.794,A -85,B 0,C 180,E1 -8378.028,E2 -8378.028} C_VEL
LIN {X 0,Y 453.208,Z 532.892,A -85,B 0,C 180,E1 -8379.371,E2 -8379.371} C_VEL
LIN {X 0,Y 453.626,Z 524.257,A -85,B 0,C 180,E1 -8380.714,E2 -8380.714} C_VEL
LIN {X 0,Y 454.179,Z 515.405,A -85,B 0,C 180,E1 -8381.831,E2 -8381.831} C_VEL
LIN {X 0,Y 454.769,Z 504.857,A -85,B 0,C 180,E1 -8382.916,E2 -8382.916} C_VEL
LIN {X 0,Y 455.239,Z 495.059,A -85,B 0,C 180,E1 -8383.731,E2 -8383.731} C_VEL
LIN {X 0,Y 455.778,Z 483.188,A -85,B 0,C 180,E1 -8384.511,E2 -8384.511} C_VEL
LIN {X 0,Y 456.247,Z 472.142,A -85,B 0,C 180,E1 -8385.067,E2 -8385.067} C_VEL
LIN {X 0,Y 454.26,Z 458.732,A -85,B 0,C 180,E1 -8385.631,E2 -8385.631} C_VEL
LIN {X 0,Y 452.858,Z 450.314,A -85,B 0,C 180,E1 -8385.901,E2 -8385.901} C_VEL
LIN {X 0,Y 453.074,Z 441.953,A -85,B 0,C 180,E1 -8389.482,E2 -8389.482} C_VEL
LIN {X 0,Y 453.266,Z 435.363,A -85,B 0,C 180,E1 -8392.326,E2 -8392.326} C_VEL
LIN {X 0,Y 453.555,Z 427.586,A -85,B 0,C 180,E1 -8395.713,E2 -8395.713} C_VEL
LIN {X 0,Y 453.903,Z 419.827,A -85,B 0,C 180,E1 -8399.191,E2 -8399.191} C_VEL
LIN {X 0,Y 454.237,Z 413.228,A -85,B 0,C 180,E1 -8402.262,E2 -8402.262} C_VEL
LIN {X 0,Y 454.522,Z 407.609,A -85,B 0,C 180,E1 -8404.964,E2 -8404.964} C_VEL
LIN {X 0,Y 454.246,Z 403.367,A -85,B 0,C 180,E1 -8407.114,E2 -8407.114} C_VEL
LIN {X 0,Y 453.53,Z 398.994,A -85,B 0,C 180,E1 -8409.518,E2 -8409.518} C_VEL
LIN {X 0,Y 453.47,Z 398.999,A -85,B 0,C 180,E1 -8412.994,E2 -8412.994} C_VEL
LIN {X 0,Y 453.468,Z 399.001,A -85,B 0,C 180,E1 -8415.779,E2 -8415.779} C_VEL
LIN {X 0,Y 453.48,Z 398.994,A -85,B 0,C 180,E1 -8418.209,E2 -8418.209} C_VEL
LIN {X 0,Y 453.512,Z 398.997,A -85,B 0,C 180,E1 -8420.791,E2 -8420.791} C_VEL
LIN {X 0,Y 453.458,Z 399,A -85,B 0,C 180,E1 -8423.917,E2 -8423.917} C_VEL
LIN {X 0,Y 453.484,Z 399,A -85,B 0,C 180,E1 -8427.151,E2 -8427.151} C_VEL
LIN {X 0,Y 453.477,Z 398.997,A -85,B 0,C 180,E1 -8430.268,E2 -8430.268} C_VEL
LIN {X 0,Y 453.506,Z 398.993,A -85,B 0,C 180,E1 -8433.294,E2 -8433.294} C_VEL
LIN {X 0,Y 453.499,Z 398.997,A -85,B 0,C 180,E1 -8436.239,E2 -8436.239} C_VEL
LIN {X 0,Y 453.485,Z 398.999,A -85,B 0,C 180,E1 -8439.118,E2 -8439.118} C_VEL
LIN {X 0,Y 453.514,Z 398.993,A -85,B 0,C 180,E1 -8441.945,E2 -8441.945} C_VEL
LIN {X 0,Y 453.542,Z 398.991,A -85,B 0,C 180,E1 -8444.726,E2 -8444.726} C_VEL
LIN {X 0,Y 453.604,Z 398.98,A -85,B 0,C 180,E1 -8447.472,E2 -8447.472} C_VEL
LIN {X 0,Y 453.595,Z 398.984,A -85,B 0,C 180,E1 -8451.087,E2 -8451.087} C_VEL
LIN {X 0,Y 453.679,Z 398.973,A -85,B 0,C 180,E1 -8453.775,E2 -8453.775} C_VEL
LIN {X 0,Y 453.746,Z 398.962,A -85,B 0,C 180,E1 -8457.337,E2 -8457.337} C_VEL
LIN {X 0,Y 453.826,Z 398.957,A -85,B 0,C 180,E1 -8460,E2 -8460} C_VEL
LIN {X 0,Y 453.745,Z 398.965,A -85,B 0,C 180,E1 -8462.663,E2 -8462.663} C_VEL
LIN {X 0,Y 453.68,Z 398.974,A -85,B 0,C 180,E1 -8466.225,E2 -8466.225} C_VEL
LIN {X 0,Y 453.595,Z 398.982,A -85,B 0,C 180,E1 -8468.913,E2 -8468.913} C_VEL
LIN {X 0,Y 453.604,Z 398.98,A -85,B 0,C 180,E1 -8472.551,E2 -8472.551} C_VEL
LIN {X 0,Y 453.546,Z 398.989,A -85,B 0,C 180,E1 -8476.196,E2 -8476.196} C_VEL
LIN {X 0,Y 453.52,Z 398.992,A -85,B 0,C 180,E1 -8479.04,E2 -8479.04} C_VEL
LIN {X 0,Y 453.478,Z 398.999,A -85,B 0,C 180,E1 -8481.836,E2 -8481.836} C_VEL
LIN {X 0,Y 453.503,Z 398.992,A -85,B 0,C 180,E1 -8484.735,E2 -8484.735} C_VEL
LIN {X 0,Y 453.539,Z 398.99,A -85,B 0,C 180,E1 -8487.961,E2 -8487.961} C_VEL
LIN {X 0,Y 453.468,Z 399,A -85,B 0,C 180,E1 -8491.525,E2 -8491.525} C_VEL
LIN {X 0,Y 453.491,Z 398.996,A -85,B 0,C 180,E1 -8494.778,E2 -8494.778} C_VEL
LIN {X 0,Y 453.475,Z 398.996,A -85,B 0,C 180,E1 -8498.311,E2 -8498.311} C_VEL
LIN {X 0,Y 453.496,Z 398.993,A -85,B 0,C 180,E1 -8500.609,E2 -8500.609} C_VEL
LIN {X 0,Y 453.458,Z 399.002,A -85,B 0,C 180,E1 -8503.244,E2 -8503.244} C_VEL
LIN {X 0,Y 453.475,Z 399,A -85,B 0,C 180,E1 -8505.78,E2 -8505.78} C_VEL
LIN {X 0,Y 453.484,Z 398.996,A -85,B 0,C 180,E1 -8508.21,E2 -8508.21} C_VEL
LIN {X 0,Y 453.496,Z 398.995,A -85,B 0,C 180,E1 -8510.794,E2 -8510.794} C_VEL
LIN {X 0,Y 453.395,Z 399.009,A -85,B 0,C 180,E1 -8513.912,E2 -8513.912} C_VEL
LIN {X 0,Y 453.369,Z 399.833,A -85,B 0,C 180,E1 -8515.245,E2 -8515.245} C_VEL
LIN {X 0,Y 453.261,Z 403.73,A -85,B 0,C 180,E1 -8518.185,E2 -8518.185} C_VEL
LIN {X 0,Y 453.148,Z 407.912,A -85,B 0,C 180,E1 -8521.263,E2 -8521.263} C_VEL
LIN {X 0,Y 453.006,Z 412.078,A -85,B 0,C 180,E1 -8524.253,E2 -8524.253} C_VEL
LIN {X 0,Y 452.862,Z 416.233,A -85,B 0,C 180,E1 -8527.171,E2 -8527.171} C_VEL
LIN {X 0,Y 452.75,Z 420.457,A -85,B 0,C 180,E1 -8530.032,E2 -8530.032} C_VEL
LIN {X 0,Y 452.7,Z 424.716,A -85,B 0,C 180,E1 -8532.844,E2 -8532.844} C_VEL
LIN {X 0,Y 452.743,Z 426.96,A -85,B 0,C 180,E1 -8534.185,E2 -8534.185} C_VEL
LIN {X 0,Y 455.466,Z 439.615,A -85,B 0,C 180,E1 -8534.657,E2 -8534.657} C_VEL
LIN {X 0,Y 456.459,Z 445.789,A -85,B 0,C 180,E1 -8534.941,E2 -8534.941} C_VEL
LIN {X 0,Y 456.081,Z 457.034,A -85,B 0,C 180,E1 -8535.499,E2 -8535.499} C_VEL
LIN {X 0,Y 455.536,Z 469.352,A -85,B 0,C 180,E1 -8536.302,E2 -8536.302} C_VEL
LIN {X 0,Y 455.08,Z 480.086,A -85,B 0,C 180,E1 -8537.208,E2 -8537.208} C_VEL
LIN {X 0,Y 454.128,Z 484.83,A -85,B 0,C 180,E1 -8537.652,E2 -8537.652} C_VEL
LIN {X 0,Y 450.853,Z 492.198,A -85,B 0,C 180,E1 -8538.392,E2 -8538.392} C_VEL
LIN {X 0,Y 447.632,Z 498.975,A -85,B 0,C 180,E1 -8539.209,E2 -8539.209} C_VEL
LIN {X 0,Y 446.76,Z 502.794,A -85,B 0,C 180,E1 -8539.764,E2 -8539.764} C_VEL
LIN {X 0,Y 446.267,Z 510.766,A -85,B 0,C 180,E1 -8541.168,E2 -8541.168} C_VEL
LIN {X 0,Y 445.837,Z 517.827,A -85,B 0,C 180,E1 -8542.755,E2 -8542.755} C_VEL
LIN {X 0,Y 445.768,Z 522.527,A -85,B 0,C 180,E1 -8544.118,E2 -8544.118} C_VEL
LIN {X 0,Y 445.501,Z 526.131,A -85,B 0,C 180,E1 -8545.476,E2 -8545.476} C_VEL
LIN {X 0,Y 445.524,Z 527.99,A -85,B 0,C 180,E1 -8546.382,E2 -8546.382} C_VEL
LIN {X 0,Y 445.464,Z 529.393,A -85,B 0,C 180,E1 -8547.287,E2 -8547.287} C_VEL
LIN {X 0,Y 445.341,Z 531.006,A -85,B 0,C 180,E1 -8549.096,E2 -8549.096} C_VEL
LIN {X 0,Y 445.342,Z 531.24,A -85,B 0,C 180,E1 -8550,E2 -8550} C_VEL
LIN {X 0,Y 445.341,Z 531.054,A -85,B 0,C 180,E1 -8550.904,E2 -8550.904} C_VEL
LIN {X 0,Y 445.463,Z 529.502,A -85,B 0,C 180,E1 -8552.713,E2 -8552.713} C_VEL
LIN {X 0,Y 445.509,Z 528.147,A -85,B 0,C 180,E1 -8553.618,E2 -8553.618} C_VEL
LIN {X 0,Y 445.54,Z 525.286,A -85,B 0,C 180,E1 -8554.977,E2 -8554.977} C_VEL
LIN {X 0,Y 445.783,Z 521.4,A -85,B 0,C 180,E1 -8556.336,E2 -8556.336} C_VEL
LIN {X 0,Y 445.958,Z 516.39,A -85,B 0,C 180,E1 -8557.698,E2 -8557.698} C_VEL
LIN {X 0,Y 446.346,Z 510.081,A -85,B 0,C 180,E1 -8559.059,E2 -8559.059} C_VEL
LIN {X 0,Y 446.768,Z 502.184,A -85,B 0,C 180,E1 -8560.423,E2 -8560.423} C_VEL
LIN {X 0,Y 447.381,Z 492.357,A -85,B 0,C 180,E1 -8561.784,E2 -8561.784} C_VEL
LIN {X 0,Y 448.078,Z 482.419,A -85,B 0,C 180,E1 -8562.878,E2 -8562.878} C_VEL
LIN {X 0,Y 448.504,Z 472.369,A -85,B 0,C 180,E1 -8563.782,E2 -8563.782} C_VEL
LIN {X 0,Y 449.097,Z 460.651,A -85,B 0,C 180,E1 -8564.616,E2 -8564.616} C_VEL
LIN {X 0,Y 449.56,Z 448.075,A -85,B 0,C 180,E1 -8565.296,E2 -8565.296} C_VEL
LIN {X 0,Y 448.939,Z 442.487,A -85,B 0,C 180,E1 -8565.562,E2 -8565.562} C_VEL
LIN {X 0,Y 446.365,Z 430.435,A -85,B 0,C 180,E1 -8566.057,E2 -8566.057} C_VEL
LIN {X 0,Y 445.589,Z 426.973,A -85,B 0,C 180,E1 -8566.185,E2 -8566.185} C_VEL
LIN {X 0,Y 445.682,Z 422.185,A -85,B 0,C 180,E1 -8569.339,E2 -8569.339} C_VEL
LIN {X 0,Y 445.762,Z 417.943,A -85,B 0,C 180,E1 -8572.234,E2 -8572.234} C_VEL
LIN {X 0,Y 445.901,Z 413.764,A -85,B 0,C 180,E1 -8575.186,E2 -8575.186} C_VEL
LIN {X 0,Y 446.036,Z 409.59,A -85,B 0,C 180,E1 -8578.21,E2 -8578.21} C_VEL
LIN {X 0,Y 446.211,Z 405.389,A -85,B 0,C 180,E1 -8581.317,E2 -8581.317} C_VEL
LIN {X 0,Y 446.308,Z 401.16,A -85,B 0,C 180,E1 -8584.534,E2 -8584.534} C_VEL
LIN {X 0,Y 446.303,Z 399.894,A -85,B 0,C 180,E1 -8585.637,E2 -8585.637} C_VEL
LIN {X 0,Y 446.415,Z 399.877,A -85,B 0,C 180,E1 -8588.079,E2 -8588.079} C_VEL
LIN {X 0,Y 446.431,Z 399.876,A -85,B 0,C 180,E1 -8590.918,E2 -8590.918} C_VEL
LIN {X 0,Y 446.424,Z 399.876,A -85,B 0,C 180,E1 -8593.843,E2 -8593.843} C_VEL
LIN {X 0,Y 446.399,Z 399.88,A -85,B 0,C 180,E1 -8596.404,E2 -8596.404} C_VEL
LIN {X 0,Y 446.43,Z 399.876,A -85,B 0,C 180,E1 -8599.082,E2 -8599.082} C_VEL
LIN {X 0,Y 446.43,Z 399.875,A -85,B 0,C 180,E1 -8602.123,E2 -8602.123} C_VEL
LIN {X 0,Y 446.432,Z 399.875,A -85,B 0,C 180,E1 -8605.477,E2 -8605.477} C_VEL
LIN {X 0,Y 446.419,Z 399.879,A -85,B 0,C 180,E1 -8608.7,E2 -8608.7} C_VEL
LIN {X 0,Y 446.488,Z 399.868,A -85,B 0,C 180,E1 -8611.821,E2 -8611.821} C_VEL
LIN {X 0,Y 446.447,Z 399.872,A -85,B 0,C 180,E1 -8614.847,E2 -8614.847} C_VEL
LIN {X 0,Y 446.451,Z 399.875,A -85,B 0,C 180,E1 -8618.245,E2 -8618.245} C_VEL
LIN {X 0,Y 446.455,Z 399.874,A -85,B 0,C 180,E1 -8621.649,E2 -8621.649} C_VEL
LIN {X 0,Y 446.511,Z 399.868,A -85,B 0,C 180,E1 -8624.48,E2 -8624.48} C_VEL
LIN {X 0,Y 446.521,Z 399.866,A -85,B 0,C 180,E1 -8628.193,E2 -8628.193} C_VEL
LIN {X 0,Y 446.604,Z 399.856,A -85,B 0,C 180,E1 -8631.858,E2 -8631.858} C_VEL
LIN {X 0,Y 446.648,Z 399.849,A -85,B 0,C 180,E1 -8634.583,E2 -8634.583} C_VEL
LIN {X 0,Y 446.667,Z 399.848,A -85,B 0,C 180,E1 -8638.197,E2 -8638.197} C_VEL
LIN {X 0,Y 446.796,Z 399.833,A -85,B 0,C 180,E1 -8640,E2 -8640} C_VEL
LIN {X 0,Y 446.694,Z 399.84,A -85,B 0,C 180,E1 -8642.705,E2 -8642.705} C_VEL
LIN {X 0,Y 446.65,Z 399.849,A -85,B 0,C 180,E1 -8646.324,E2 -8646.324} C_VEL
LIN {X 0,Y 446.542,Z 399.863,A -85,B 0,C 180,E1 -8649.055,E2 -8649.055} C_VEL
LIN {X 0,Y 446.537,Z 399.861,A -85,B 0,C 180,E1 -8652.729,E2 -8652.729} C_VEL
LIN {X 0,Y 446.493,Z 399.865,A -85,B 0,C 180,E1 -8656.459,E2 -8656.459} C_VEL
LIN {X 0,Y 446.473,Z 399.872,A -85,B 0,C 180,E1 -8659.303,E2 -8659.303} C_VEL
LIN {X 0,Y 446.42,Z 399.876,A -85,B 0,C 180,E1 -8662.2,E2 -8662.2} C_VEL
LIN {X 0,Y 446.447,Z 399.874,A -85,B 0,C 180,E1 -8665.153,E2 -8665.153} C_VEL
LIN {X 0,Y 446.487,Z 399.865,A -85,B 0,C 180,E1 -8668.179,E2 -8668.179} C_VEL
LIN {X 0,Y 446.422,Z 399.876,A -85,B 0,C 180,E1 -8671.775,E2 -8671.775} C_VEL
LIN {X 0,Y 446.433,Z 399.876,A -85,B 0,C 180,E1 -8674.523,E2 -8674.523} C_VEL
LIN {X 0,Y 446.433,Z 399.874,A -85,B 0,C 180,E1 -8678.082,E2 -8678.082} C_VEL
LIN {X 0,Y 446.43,Z 399.878,A -85,B 0,C 180,E1 -8680.918,E2 -8680.918} C_VEL
LIN {X 0,Y 446.404,Z 399.878,A -85,B 0,C 180,E1 -8683.846,E2 -8683.846} C_VEL
LIN {X 0,Y 446.423,Z 399.881,A -85,B 0,C 180,E1 -8686.4,E2 -8686.4} C_VEL
LIN {X 0,Y 446.468,Z 399.877,A -85,B 0,C 180,E1 -8689.805,E2 -8689.805} C_VEL
LIN {X 0,Y 446.502,Z 399.988,A -85,B 0,C 180,E1 -8690.364,E2 -8690.364} C_VEL
LIN {X 0,Y 447.374,Z 405.493,A -85,B 0,C 180,E1 -8693.347,E2 -8693.347} C_VEL
LIN {X 0,Y 447.475,Z 409.847,A -85,B 0,C 180,E1 -8695.569,E2 -8695.569} C_VEL
LIN {X 0,Y 447.094,Z 416.428,A -85,B 0,C 180,E1 -8698.752,E2 -8698.752} C_VEL
LIN {X 0,Y 446.853,Z 421.938,A -85,B 0,C 180,E1 -8701.335,E2 -8701.335} C_VEL
LIN {X 0,Y 446.455,Z 429.686,A -85,B 0,C 180,E1 -8704.847,E2 -8704.847} C_VEL
LIN {X 0,Y 446.181,Z 437.535,A -85,B 0,C 180,E1 -8708.332,E2 -8708.332} C_VEL
LIN {X 0,Y 445.892,Z 445.067,A -85,B 0,C 180,E1 -8711.625,E2 -8711.625} C_VEL
LIN {X 0,Y 445.776,Z 450.152,A -85,B 0,C 180,E1 -8713.85,E2 -8713.85} C_VEL
LIN {X 0,Y 447.996,Z 463.265,A -85,B 0,C 180,E1 -8714.295,E2 -8714.295} C_VEL
LIN {X 0,Y 449.298,Z 474.494,A -85,B 0,C 180,E1 -8714.811,E2 -8714.811} C_VEL
LIN {X 0,Y 448.734,Z 486.704,A -85,B 0,C 180,E1 -8715.487,E2 -8715.487} C_VEL
LIN {X 0,Y 448.049,Z 499.151,A -85,B 0,C 180,E1 -8716.391,E2 -8716.391} C_VEL
LIN {X 0,Y 447.507,Z 510.063,A -85,B 0,C 180,E1 -8717.414,E2 -8717.414} C_VEL
LIN {X 0,Y 447,Z 518.962,A -85,B 0,C 180,E1 -8718.436,E2 -8718.436} C_VEL
LIN {X 0,Y 446.426,Z 527.138,A -85,B 0,C 180,E1 -8719.569,E2 -8719.569} C_VEL
LIN {X 0,Y 446.032,Z 535.167,A -85,B 0,C 180,E1 -8720.934,E2 -8720.934} C_VEL
LIN {X 0,Y 445.742,Z 541.605,A -85,B 0,C 180,E1 -8722.298,E2 -8722.298} C_VEL
LIN {X 0,Y 445.492,Z 547.562,A -85,B 0,C 180,E1 -8723.928,E2 -8723.928} C_VEL
LIN {X 0,Y 445.417,Z 551.761,A -85,B 0,C 180,E1 -8725.475,E2 -8725.475} C_VEL
LIN {X 0,Y 445.381,Z 553.623,A -85,B 0,C 180,E1 -8726.381,E2 -8726.381} C_VEL
LIN {X 0,Y 445.433,Z 555.021,A -85,B 0,C 180,E1 -8727.287,E2 -8727.287} C_VEL
LIN {X 0,Y 445.338,Z 556.623,A -85,B 0,C 180,E1 -8729.096,E2 -8729.096} C_VEL
LIN {X 0,Y 445.342,Z 556.84,A -85,B 0,C 180,E1 -8730,E2 -8730} C_VEL
LIN {X 0,Y 445.338,Z 556.623,A -85,B 0,C 180,E1 -8730.904,E2 -8730.904} C_VEL
LIN {X 0,Y 445.433,Z 555.023,A -85,B 0,C 180,E1 -8732.713,E2 -8732.713} C_VEL
LIN {X 0,Y 445.381,Z 553.624,A -85,B 0,C 180,E1 -8733.619,E2 -8733.619} C_VEL
LIN {X 0,Y 445.479,Z 550.689,A -85,B 0,C 180,E1 -8734.978,E2 -8734.978} C_VEL
LIN {X 0,Y 445.576,Z 545.281,A -85,B 0,C 180,E1 -8736.748,E2 -8736.748} C_VEL
LIN {X 0,Y 445.847,Z 539.589,A -85,B 0,C 180,E1 -8738.156,E2 -8738.156} C_VEL
LIN {X 0,Y 446.157,Z 532.685,A -85,B 0,C 180,E1 -8739.52,E2 -8739.52} C_VEL
LIN {X 0,Y 446.617,Z 524.05,A -85,B 0,C 180,E1 -8740.885,E2 -8740.885} C_VEL
LIN {X 0,Y 447.206,Z 515.198,A -85,B 0,C 180,E1 -8742.018,E2 -8742.018} C_VEL
LIN {X 0,Y 447.826,Z 504.298,A -85,B 0,C 180,E1 -8743.154,E2 -8743.154} C_VEL
LIN {X 0,Y 448.333,Z 494.851,A -85,B 0,C 180,E1 -8743.946,E2 -8743.946} C_VEL
LIN {X 0,Y 448.885,Z 482.979,A -85,B 0,C 180,E1 -8744.739,E2 -8744.739} C_VEL
LIN {X 0,Y 449.356,Z 473.234,A -85,B 0,C 180,E1 -8745.245,E2 -8745.245} C_VEL
LIN {X 0,Y 447.438,Z 459.761,A -85,B 0,C 180,E1 -8745.836,E2 -8745.836} C_VEL
LIN {X 0,Y 445.774,Z 450.104,A -85,B 0,C 180,E1 -8746.165,E2 -8746.165} C_VEL
LIN {X 0,Y 446.032,Z 441.778,A -85,B 0,C 180,E1 -8749.802,E2 -8749.802} C_VEL
LIN {X 0,Y 446.224,Z 435.203,A -85,B 0,C 180,E1 -8752.698,E2 -8752.698} C_VEL
LIN {X 0,Y 446.49,Z 428.55,A -85,B 0,C 180,E1 -8755.65,E2 -8755.65} C_VEL
LIN {X 0,Y 446.873,Z 420.811,A -85,B 0,C 180,E1 -8759.179,E2 -8759.179} C_VEL
LIN {X 0,Y 447.212,Z 414.215,A -85,B 0,C 180,E1 -8762.297,E2 -8762.297} C_VEL
LIN {X 0,Y 447.526,Z 408.19,A -85,B 0,C 180,E1 -8765.253,E2 -8765.253} C_VEL
LIN {X 0,Y 447.341,Z 405.278,A -85,B 0,C 180,E1 -8766.751,E2 -8766.751} C_VEL
LIN {X 0,Y 446.488,Z 399.871,A -85,B 0,C 180,E1 -8769.728,E2 -8769.728} C_VEL
LIN {X 0,Y 446.434,Z 399.876,A -85,B 0,C 180,E1 -8772.604,E2 -8772.604} C_VEL
LIN {X 0,Y 446.456,Z 399.874,A -85,B 0,C 180,E1 -8775.103,E2 -8775.103} C_VEL
LIN {X 0,Y 446.429,Z 399.875,A -85,B 0,C 180,E1 -8778.609,E2 -8778.609} C_VEL
LIN {X 0,Y 446.459,Z 399.874,A -85,B 0,C 180,E1 -8780.974,E2 -8780.974} C_VEL
LIN {X 0,Y 446.423,Z 399.878,A -85,B 0,C 180,E1 -8784.374,E2 -8784.374} C_VEL
LIN {X 0,Y 446.424,Z 399.876,A -85,B 0,C 180,E1 -8787.638,E2 -8787.638} C_VEL
LIN {X 0,Y 446.451,Z 399.876,A -85,B 0,C 180,E1 -8790.791,E2 -8790.791} C_VEL
LIN {X 0,Y 446.479,Z 399.868,A -85,B 0,C 180,E1 -8793.848,E2 -8793.848} C_VEL
LIN {X 0,Y 446.428,Z 399.877,A -85,B 0,C 180,E1 -8796.823,E2 -8796.823} C_VEL
LIN {X 0,Y 446.447,Z 399.873,A -85,B 0,C 180,E1 -8799.737,E2 -8799.737} C_VEL
LIN {X 0,Y 446.466,Z 399.874,A -85,B 0,C 180,E1 -8802.597,E2 -8802.597} C_VEL
LIN {X 0,Y 446.472,Z 399.867,A -85,B 0,C 180,E1 -8805.412,E2 -8805.412} C_VEL
LIN {X 0,Y 446.541,Z 399.865,A -85,B 0,C 180,E1 -8808.194,E2 -8808.194} C_VEL
LIN {X 0,Y 446.602,Z 399.855,A -85,B 0,C 180,E1 -8811.858,E2 -8811.858} C_VEL
LIN {X 0,Y 446.647,Z 399.852,A -85,B 0,C 180,E1 -8814.583,E2 -8814.583} C_VEL
LIN {X 0,Y 446.666,Z 399.849,A -85,B 0,C 180,E1 -8818.197,E2 -8818.197} C_VEL
LIN {X 0,Y 446.796,Z 399.832,A -85,B 0,C 180,E1 -8820,E2 -8820} C_VEL
LIN {X 0,Y 446.692,Z 399.843,A -85,B 0,C 180,E1 -8822.705,E2 -8822.705} C_VEL
LIN {X 0,Y 446.649,Z 399.85,A -85,B 0,C 180,E1 -8826.324,E2 -8826.324} C_VEL
LIN {X 0,Y 446.541,Z 399.86,A -85,B 0,C 180,E1 -8829.055,E2 -8829.055} C_VEL
LIN {X 0,Y 446.536,Z 399.86,A -85,B 0,C 180,E1 -8832.729,E2 -8832.729} C_VEL
LIN {X 0,Y 446.49,Z 399.869,A -85,B 0,C 180,E1 -8836.459,E2 -8836.459} C_VEL
LIN {X 0,Y 446.47,Z 399.872,A -85,B 0,C 180,E1 -8839.303,E2 -8839.303} C_VEL
LIN {X 0,Y 446.42,Z 399.878,A -85,B 0,C 180,E1 -8842.2,E2 -8842.2} C_VEL
LIN {X 0,Y 446.446,Z 399.872,A -85,B 0,C 180,E1 -8845.153,E2 -8845.153} C_VEL
LIN {X 0,Y 446.486,Z 399.868,A -85,B 0,C 180,E1 -8848.179,E2 -8848.179} C_VEL
LIN {X 0,Y 446.421,Z 399.878,A -85,B 0,C 180,E1 -8851.775,E2 -8851.775} C_VEL
LIN {X 0,Y 446.433,Z 399.875,A -85,B 0,C 180,E1 -8854.523,E2 -8854.523} C_VEL
LIN {X 0,Y 446.433,Z 399.874,A -85,B 0,C 180,E1 -8858.082,E2 -8858.082} C_VEL
LIN {X 0,Y 446.429,Z 399.875,A -85,B 0,C 180,E1 -8860.918,E2 -8860.918} C_VEL
LIN {X 0,Y 446.404,Z 399.879,A -85,B 0,C 180,E1 -8863.846,E2 -8863.846} C_VEL
LIN {X 0,Y 446.423,Z 399.876,A -85,B 0,C 180,E1 -8866.4,E2 -8866.4} C_VEL
LIN {X 0,Y 446.445,Z 399.874,A -85,B 0,C 180,E1 -8869.802,E2 -8869.802} C_VEL
LIN {X 0,Y 446.407,Z 399.877,A -85,B 0,C 180,E1 -8872.121,E2 -8872.121} C_VEL
LIN {X 0,Y 446.301,Z 399.894,A -85,B 0,C 180,E1 -8874.363,E2 -8874.363} C_VEL
LIN {X 0,Y 446.309,Z 401.03,A -85,B 0,C 180,E1 -8875.466,E2 -8875.466} C_VEL
LIN {X 0,Y 446.209,Z 405.247,A -85,B 0,C 180,E1 -8878.684,E2 -8878.684} C_VEL
LIN {X 0,Y 446.031,Z 409.447,A -85,B 0,C 180,E1 -8881.79,E2 -8881.79} C_VEL
LIN {X 0,Y 445.902,Z 413.622,A -85,B 0,C 180,E1 -8884.814,E2 -8884.814} C_VEL
LIN {X 0,Y 445.762,Z 417.801,A -85,B 0,C 180,E1 -8887.766,E2 -8887.766} C_VEL
LIN {X 0,Y 445.713,Z 422.685,A -85,B 0,C 180,E1 -8891.1,E2 -8891.1} C_VEL
LIN {X 0,Y 445.648,Z 426.965,A -85,B 0,C 180,E1 -8893.907,E2 -8893.907} C_VEL
LIN {X 0,Y 448.832,Z 441.979,A -85,B 0,C 180,E1 -8894.507,E2 -8894.507} C_VEL
LIN {X 0,Y 449.604,Z 447.3,A -85,B 0,C 180,E1 -8894.763,E2 -8894.763} C_VEL
LIN {X 0,Y 449.154,Z 459.222,A -85,B 0,C 180,E1 -8895.386,E2 -8895.386} C_VEL
LIN {X 0,Y 448.578,Z 470.986,A -85,B 0,C 180,E1 -8896.2,E2 -8896.2} C_VEL
LIN {X 0,Y 448.022,Z 482.376,A -85,B 0,C 180,E1 -8897.208,E2 -8897.208} C_VEL
LIN {X 0,Y 447.416,Z 491.61,A -85,B 0,C 180,E1 -8898.217,E2 -8898.217} C_VEL
LIN {X 0,Y 446.951,Z 500.11,A -85,B 0,C 180,E1 -8899.353,E2 -8899.353} C_VEL
LIN {X 0,Y 446.76,Z 502.794,A -85,B 0,C 180,E1 -8899.764,E2 -8899.764} C_VEL
LIN {X 0,Y 445.886,Z 506.471,A -85,B 0,C 180,E1 -8900.347,E2 -8900.347} C_VEL
LIN {X 0,Y 442.67,Z 511.994,A -85,B 0,C 180,E1 -8901.326,E2 -8901.326} C_VEL
LIN {X 0,Y 439.507,Z 516.936,A -85,B 0,C 180,E1 -8902.372,E2 -8902.372} C_VEL
LIN {X 0,Y 438.726,Z 519.558,A -85,B 0,C 180,E1 -8903.053,E2 -8903.053} C_VEL
LIN {X 0,Y 438.602,Z 524.048,A -85,B 0,C 180,E1 -8904.483,E2 -8904.483} C_VEL
LIN {X 0,Y 438.424,Z 526.336,A -85,B 0,C 180,E1 -8905.403,E2 -8905.403} C_VEL
LIN {X 0,Y 438.428,Z 528.195,A -85,B 0,C 180,E1 -8906.324,E2 -8906.324} C_VEL
LIN {X 0,Y 438.395,Z 529.597,A -85,B 0,C 180,E1 -8907.243,E2 -8907.243} C_VEL
LIN {X 0,Y 438.255,Z 531.21,A -85,B 0,C 180,E1 -8909.081,E2 -8909.081} C_VEL
LIN {X 0,Y 438.254,Z 531.444,A -85,B 0,C 180,E1 -8910,E2 -8910} C_VEL
LIN {X 0,Y 438.255,Z 531.257,A -85,B 0,C 180,E1 -8910.919,E2 -8910.919} C_VEL
LIN {X 0,Y 438.393,Z 529.705,A -85,B 0,C 180,E1 -8912.757,E2 -8912.757} C_VEL
LIN {X 0,Y 438.413,Z 528.351,A -85,B 0,C 180,E1 -8913.677,E2 -8913.677} C_VEL
LIN {X 0,Y 438.482,Z 525.488,A -85,B 0,C 180,E1 -8915.058,E2 -8915.058} C_VEL
LIN {X 0,Y 438.705,Z 520.856,A -85,B 0,C 180,E1 -8916.668,E2 -8916.668} C_VEL
LIN {X 0,Y 439.011,Z 514.622,A -85,B 0,C 180,E1 -8918.284,E2 -8918.284} C_VEL
LIN {X 0,Y 439.465,Z 507.836,A -85,B 0,C 180,E1 -8919.667,E2 -8919.667} C_VEL
LIN {X 0,Y 439.931,Z 500.905,A -85,B 0,C 180,E1 -8920.819,E2 -8920.819} C_VEL
LIN {X 0,Y 440.435,Z 492.557,A -85,B 0,C 180,E1 -8921.973,E2 -8921.973} C_VEL
LIN {X 0,Y 441.146,Z 482.768,A -85,B 0,C 180,E1 -8923.069,E2 -8923.069} C_VEL
LIN {X 0,Y 441.648,Z 472.027,A -85,B 0,C 180,E1 -8924.045,E2 -8924.045} C_VEL
LIN {X 0,Y 442.228,Z 460.848,A -85,B 0,C 180,E1 -8924.849,E2 -8924.849} C_VEL
LIN {X 0,Y 442.716,Z 448.269,A -85,B 0,C 180,E1 -8925.539,E2 -8925.539} C_VEL
LIN {X 0,Y 440.874,Z 437.15,A -85,B 0,C 180,E1 -8926.063,E2 -8926.063} C_VEL
LIN {X 0,Y 438.518,Z 427.165,A -85,B 0,C 180,E1 -8926.452,E2 -8926.452} C_VEL
LIN {X 0,Y 438.623,Z 422.364,A -85,B 0,C 180,E1 -8929.663,E2 -8929.663} C_VEL
LIN {X 0,Y 438.704,Z 418.108,A -85,B 0,C 180,E1 -8932.612,E2 -8932.612} C_VEL
LIN {X 0,Y 438.857,Z 413.917,A -85,B 0,C 180,E1 -8935.619,E2 -8935.619} C_VEL
LIN {X 0,Y 439.013,Z 409.724,A -85,B 0,C 180,E1 -8938.703,E2 -8938.703} C_VEL
LIN {X 0,Y 439.186,Z 405.51,A -85,B 0,C 180,E1 -8941.876,E2 -8941.876} C_VEL
LIN {X 0,Y 439.246,Z 402.677,A -85,B 0,C 180,E1 -8944.056,E2 -8944.056} C_VEL
LIN {X 0,Y 439.261,Z 401.082,A -85,B 0,C 180,E1 -8945.315,E2 -8945.315} C_VEL
LIN {X 0,Y 439.341,Z 400.757,A -85,B 0,C 180,E1 -8947.436,E2 -8947.436} C_VEL
LIN {X 0,Y 439.404,Z 400.749,A -85,B 0,C 180,E1 -8949.849,E2 -8949.849} C_VEL
LIN {X 0,Y 439.388,Z 400.755,A -85,B 0,C 180,E1 -8952.627,E2 -8952.627} C_VEL
LIN {X 0,Y 439.403,Z 400.752,A -85,B 0,C 180,E1 -8955.271,E2 -8955.271} C_VEL
LIN {X 0,Y 439.391,Z 400.756,A -85,B 0,C 180,E1 -8958.743,E2 -8958.743} C_VEL
LIN {X 0,Y 439.387,Z 400.75,A -85,B 0,C 180,E1 -8961.606,E2 -8961.606} C_VEL
LIN {X 0,Y 439.402,Z 400.751,A -85,B 0,C 180,E1 -8964.844,E2 -8964.844} C_VEL
LIN {X 0,Y 439.376,Z 400.756,A -85,B 0,C 180,E1 -8968.14,E2 -8968.14} C_VEL
LIN {X 0,Y 439.435,Z 400.746,A -85,B 0,C 180,E1 -8971.598,E2 -8971.598} C_VEL
LIN {X 0,Y 439.401,Z 400.754,A -85,B 0,C 180,E1 -8974.415,E2 -8974.415} C_VEL
LIN {X 0,Y 439.367,Z 400.754,A -85,B 0,C 180,E1 -8977.425,E2 -8977.425} C_VEL
LIN {X 0,Y 439.444,Z 400.747,A -85,B 0,C 180,E1 -8980.663,E2 -8980.663} C_VEL
LIN {X 0,Y 439.465,Z 400.745,A -85,B 0,C 180,E1 -8984.225,E2 -8984.225} C_VEL
LIN {X 0,Y 439.487,Z 400.743,A -85,B 0,C 180,E1 -8988.001,E2 -8988.001} C_VEL
LIN {X 0,Y 439.551,Z 400.735,A -85,B 0,C 180,E1 -8991.726,E2 -8991.726} C_VEL
LIN {X 0,Y 439.624,Z 400.724,A -85,B 0,C 180,E1 -8994.496,E2 -8994.496} C_VEL
LIN {X 0,Y 439.637,Z 400.724,A -85,B 0,C 180,E1 -8998.168,E2 -8998.168} C_VEL
LIN {X 0,Y 439.766,Z 400.708,A -85,B 0,C 180,E1 -9000,E2 -9000} C_VEL
LIN {X 0,Y 439.644,Z 400.718,A -85,B 0,C 180,E1 -9002.749,E2 -9002.749} C_VEL
LIN {X 0,Y 439.621,Z 400.723,A -85,B 0,C 180,E1 -9006.425,E2 -9006.425} C_VEL
LIN {X 0,Y 439.504,Z 400.74,A -85,B 0,C 180,E1 -9009.202,E2 -9009.202} C_VEL
LIN {X 0,Y 439.507,Z 400.736,A -85,B 0,C 180,E1 -9012.726,E2 -9012.726} C_VEL
LIN {X 0,Y 439.451,Z 400.743,A -85,B 0,C 180,E1 -9016.349,E2 -9016.349} C_VEL
LIN {X 0,Y 439.406,Z 400.751,A -85,B 0,C 180,E1 -9019.626,E2 -9019.626} C_VEL
LIN {X 0,Y 439.367,Z 400.755,A -85,B 0,C 180,E1 -9022.575,E2 -9022.575} C_VEL
LIN {X 0,Y 439.401,Z 400.753,A -85,B 0,C 180,E1 -9025.585,E2 -9025.585} C_VEL
LIN {X 0,Y 439.42,Z 400.747,A -85,B 0,C 180,E1 -9028.673,E2 -9028.673} C_VEL
LIN {X 0,Y 439.373,Z 400.753,A -85,B 0,C 180,E1 -9032.03,E2 -9032.03} C_VEL
LIN {X 0,Y 439.398,Z 400.753,A -85,B 0,C 180,E1 -9035.341,E2 -9035.341} C_VEL
LIN {X 0,Y 439.391,Z 400.753,A -85,B 0,C 180,E1 -9038.594,E2 -9038.594} C_VEL
LIN {X 0,Y 439.391,Z 400.753,A -85,B 0,C 180,E1 -9041.257,E2 -9041.257} C_VEL
LIN {X 0,Y 439.405,Z 400.754,A -85,B 0,C 180,E1 -9044.729,E2 -9044.729} C_VEL
LIN {X 0,Y 439.4,Z 400.756,A -85,B 0,C 180,E1 -9047.796,E2 -9047.796} C_VEL
LIN {X 0,Y 439.466,Z 400.888,A -85,B 0,C 180,E1 -9050.141,E2 -9050.141} C_VEL
LIN {X 0,Y 440.269,Z 405.946,A -85,B 0,C 180,E1 -9052.954,E2 -9052.954} C_VEL
LIN {X 0,Y 440.507,Z 409.758,A -85,B 0,C 180,E1 -9054.945,E2 -9054.945} C_VEL
LIN {X 0,Y 440.123,Z 416.312,A -85,B 0,C 180,E1 -9058.2,E2 -9058.2} C_VEL
LIN {X 0,Y 439.859,Z 421.809,A -85,B 0,C 180,E1 -9060.835,E2 -9060.835} C_VEL
LIN {X 0,Y 439.426,Z 429.538,A -85,B 0,C 180,E1 -9064.416,E2 -9064.416} C_VEL
LIN {X 0,Y 439.178,Z 436.148,A -85,B 0,C 180,E1 -9067.414,E2 -9067.414} C_VEL
LIN {X 0,Y 438.948,Z 442.707,A -85,B 0,C 180,E1 -9070.352,E2 -9070.352} C_VEL
LIN {X 0,Y 438.709,Z 449.909,A -85,B 0,C 180,E1 -9073.566,E2 -9073.566} C_VEL
LIN {X 0,Y 441.193,Z 464.822,A -85,B 0,C 180,E1 -9074.114,E2 -9074.114} C_VEL
LIN {X 0,Y 442.38,Z 475.426,A -85,B 0,C 180,E1 -9074.626,E2 -9074.626} C_VEL
LIN {X 0,Y 441.755,Z 488.272,A -85,B 0,C 180,E1 -9075.371,E2 -9075.371} C_VEL
LIN {X 0,Y 441.143,Z 498.95,A -85,B 0,C 180,E1 -9076.174,E2 -9076.174} C_VEL
LIN {X 0,Y 440.526,Z 509.86,A -85,B 0,C 180,E1 -9077.211,E2 -9077.211} C_VEL
LIN {X 0,Y 440.007,Z 518.759,A -85,B 0,C 180,E1 -9078.249,E2 -9078.249} C_VEL
LIN {X 0,Y 439.344,Z 528.426,A -85,B 0,C 180,E1 -9079.632,E2 -9079.632} C_VEL
LIN {X 0,Y 438.938,Z 536.125,A -85,B 0,C 180,E1 -9081.019,E2 -9081.019} C_VEL
LIN {X 0,Y 438.607,Z 543.224,A -85,B 0,C 180,E1 -9082.635,E2 -9082.635} C_VEL
LIN {X 0,Y 438.392,Z 547.79,A -85,B 0,C 180,E1 -9083.968,E2 -9083.968} C_VEL
LIN {X 0,Y 438.346,Z 551.557,A -85,B 0,C 180,E1 -9085.402,E2 -9085.402} C_VEL
LIN {X 0,Y 438.283,Z 553.419,A -85,B 0,C 180,E1 -9086.322,E2 -9086.322} C_VEL
LIN {X 0,Y 438.341,Z 554.817,A -85,B 0,C 180,E1 -9087.243,E2 -9087.243} C_VEL
LIN {X 0,Y 438.252,Z 556.42,A -85,B 0,C 180,E1 -9089.081,E2 -9089.081} C_VEL
LIN {X 0,Y 438.253,Z 556.636,A -85,B 0,C 180,E1 -9090,E2 -9090} C_VEL
LIN {X 0,Y 438.278,Z 555.813,A -85,B 0,C 180,E1 -9091.838,E2 -9091.838} C_VEL
LIN {X 0,Y 438.341,Z 554.818,A -85,B 0,C 180,E1 -9092.757,E2 -9092.757} C_VEL
LIN {X 0,Y 438.283,Z 553.419,A -85,B 0,C 180,E1 -9093.677,E2 -9093.677} C_VEL
LIN {X 0,Y 438.39,Z 550.484,A -85,B 0,C 180,E1 -9095.058,E2 -9095.058} C_VEL
LIN {X 0,Y 438.449,Z 546.507,A -85,B 0,C 180,E1 -9096.442,E2 -9096.442} C_VEL
LIN {X 0,Y 438.723,Z 540.395,A -85,B 0,C 180,E1 -9098.058,E2 -9098.058} C_VEL
LIN {X 0,Y 439.064,Z 533.716,A -85,B 0,C 180,E1 -9099.443,E2 -9099.443} C_VEL
LIN {X 0,Y 439.524,Z 525.431,A -85,B 0,C 180,E1 -9100.829,E2 -9100.829} C_VEL
LIN {X 0,Y 440.116,Z 516.942,A -85,B 0,C 180,E1 -9101.981,E2 -9101.981} C_VEL
LIN {X 0,Y 440.746,Z 506.835,A -85,B 0,C 180,E1 -9103.096,E2 -9103.096} C_VEL
LIN {X 0,Y 441.324,Z 496.072,A -85,B 0,C 180,E1 -9104.055,E2 -9104.055} C_VEL
LIN {X 0,Y 441.939,Z 484.696,A -85,B 0,C 180,E1 -9104.858,E2 -9104.858} C_VEL
LIN {X 0,Y 442.454,Z 474.237,A -85,B 0,C 180,E1 -9105.43,E2 -9105.43} C_VEL
LIN {X 0,Y 440.66,Z 461.051,A -85,B 0,C 180,E1 -9106.037,E2 -9106.037} C_VEL
LIN {X 0,Y 438.709,Z 449.904,A -85,B 0,C 180,E1 -9106.434,E2 -9106.434} C_VEL
LIN {X 0,Y 438.95,Z 442.697,A -85,B 0,C 180,E1 -9109.647,E2 -9109.647} C_VEL
LIN {X 0,Y 439.17,Z 436.132,A -85,B 0,C 180,E1 -9112.586,E2 -9112.586} C_VEL
LIN {X 0,Y 439.424,Z 429.515,A -85,B 0,C 180,E1 -9115.584,E2 -9115.584} C_VEL
LIN {X 0,Y 439.853,Z 421.787,A -85,B 0,C 180,E1 -9119.165,E2 -9119.165} C_VEL
LIN {X 0,Y 440.17,Z 415.476,A -85,B 0,C 180,E1 -9122.196,E2 -9122.196} C_VEL
LIN {X 0,Y 440.504,Z 409.73,A -85,B 0,C 180,E1 -9125.055,E2 -9125.055} C_VEL
LIN {X 0,Y 440.17,Z 405.391,A -85,B 0,C 180,E1 -9127.353,E2 -9127.353} C_VEL
LIN {X 0,Y 439.464,Z 400.747,A -85,B 0,C 180,E1 -9129.965,E2 -9129.965} C_VEL
LIN {X 0,Y 439.371,Z 400.758,A -85,B 0,C 180,E1 -9133.457,E2 -9133.457} C_VEL
LIN {X 0,Y 439.353,Z 400.756,A -85,B 0,C 180,E1 -9136.541,E2 -9136.541} C_VEL
LIN {X 0,Y 439.382,Z 400.756,A -85,B 0,C 180,E1 -9139.019,E2 -9139.019} C_VEL
LIN {X 0,Y 439.386,Z 400.753,A -85,B 0,C 180,E1 -9141.606,E2 -9141.606} C_VEL
LIN {X 0,Y 439.402,Z 400.752,A -85,B 0,C 180,E1 -9144.844,E2 -9144.844} C_VEL
LIN {X 0,Y 439.374,Z 400.754,A -85,B 0,C 180,E1 -9148.14,E2 -9148.14} C_VEL
LIN {X 0,Y 439.434,Z 400.744,A -85,B 0,C 180,E1 -9151.598,E2 -9151.598} C_VEL
LIN {X 0,Y 439.399,Z 400.753,A -85,B 0,C 180,E1 -9154.415,E2 -9154.415} C_VEL
LIN {X 0,Y 439.365,Z 400.755,A -85,B 0,C 180,E1 -9157.425,E2 -9157.425} C_VEL
LIN {X 0,Y 439.443,Z 400.748,A -85,B 0,C 180,E1 -9160.663,E2 -9160.663} C_VEL
LIN {X 0,Y 439.464,Z 400.743,A -85,B 0,C 180,E1 -9164.225,E2 -9164.225} C_VEL
LIN {X 0,Y 439.51,Z 400.738,A -85,B 0,C 180,E1 -9168.002,E2 -9168.002} C_VEL
LIN {X 0,Y 439.55,Z 400.733,A -85,B 0,C 180,E1 -9171.726,E2 -9171.726} C_VEL
LIN {X 0,Y 439.623,Z 400.726,A -85,B 0,C 180,E1 -9174.496,E2 -9174.496} C_VEL
LIN {X 0,Y 439.636,Z 400.724,A -85,B 0,C 180,E1 -9178.168,E2 -9178.168} C_VEL
LIN {X 0,Y 439.766,Z 400.708,A -85,B 0,C 180,E1 -9180,E2 -9180} C_VEL
LIN {X 0,Y 439.642,Z 400.722,A -85,B 0,C 180,E1 -9182.749,E2 -9182.749} C_VEL
LIN {X 0,Y 439.62,Z 400.726,A -85,B 0,C 180,E1 -9186.425,E2 -9186.425} C_VEL
LIN {X 0,Y 439.503,Z 400.737,A -85,B 0,C 180,E1 -9189.202,E2 -9189.202} C_VEL
LIN {X 0,Y 439.506,Z 400.736,A -85,B 0,C 180,E1 -9192.727,E2 -9192.727} C_VEL
LIN {X 0,Y 439.448,Z 400.746,A -85,B 0,C 180,E1 -9196.348,E2 -9196.348} C_VEL
LIN {X 0,Y 439.404,Z 400.752,A -85,B 0,C 180,E1 -9199.626,E2 -9199.626} C_VEL
LIN {X 0,Y 439.366,Z 400.754,A -85,B 0,C 180,E1 -9202.576,E2 -9202.576} C_VEL
LIN {X 0,Y 439.4,Z 400.753,A -85,B 0,C 180,E1 -9205.585,E2 -9205.585} C_VEL
LIN {X 0,Y 439.419,Z 400.747,A -85,B 0,C 180,E1 -9208.673,E2 -9208.673} C_VEL
LIN {X 0,Y 439.372,Z 400.757,A -85,B 0,C 180,E1 -9212.031,E2 -9212.031} C_VEL
LIN {X 0,Y 439.399,Z 400.752,A -85,B 0,C 180,E1 -9215.341,E2 -9215.341} C_VEL
LIN {X 0,Y 439.392,Z 400.75,A -85,B 0,C 180,E1 -9218.594,E2 -9218.594} C_VEL
LIN {X 0,Y 439.39,Z 400.756,A -85,B 0,C 180,E1 -9221.257,E2 -9221.257} C_VEL
LIN {X 0,Y 439.404,Z 400.751,A -85,B 0,C 180,E1 -9224.729,E2 -9224.729} C_VEL
LIN {X 0,Y 439.4,Z 400.752,A -85,B 0,C 180,E1 -9227.796,E2 -9227.796} C_VEL
LIN {X 0,Y 439.428,Z 400.746,A -85,B 0,C 180,E1 -9230.227,E2 -9230.227} C_VEL
LIN {X 0,Y 439.302,Z 400.765,A -85,B 0,C 180,E1 -9233.706,E2 -9233.706} C_VEL
LIN {X 0,Y 439.258,Z 401.136,A -85,B 0,C 180,E1 -9234.831,E2 -9234.831} C_VEL
LIN {X 0,Y 439.22,Z 403.963,A -85,B 0,C 180,E1 -9237.041,E2 -9237.041} C_VEL
LIN {X 0,Y 439.089,Z 408.174,A -85,B 0,C 180,E1 -9240.252,E2 -9240.252} C_VEL
LIN {X 0,Y 438.908,Z 412.874,A -85,B 0,C 180,E1 -9243.728,E2 -9243.728} C_VEL
LIN {X 0,Y 438.773,Z 416.553,A -85,B 0,C 180,E1 -9246.395,E2 -9246.395} C_VEL
LIN {X 0,Y 438.627,Z 420.806,A -85,B 0,C 180,E1 -9249.36,E2 -9249.36} C_VEL
LIN {X 0,Y 438.576,Z 425.093,A -85,B 0,C 180,E1 -9252.274,E2 -9252.274} C_VEL
LIN {X 0,Y 438.561,Z 427.169,A -85,B 0,C 180,E1 -9253.647,E2 -9253.647} C_VEL
LIN {X 0,Y 441.646,Z 441.149,A -85,B 0,C 180,E1 -9254.208,E2 -9254.208} C_VEL
LIN {X 0,Y 442.721,Z 447.515,A -85,B 0,C 180,E1 -9254.521,E2 -9254.521} C_VEL
LIN {X 0,Y 442.283,Z 459.434,A -85,B 0,C 180,E1 -9255.154,E2 -9255.154} C_VEL
LIN {X 0,Y 441.676,Z 471.196,A -85,B 0,C 180,E1 -9255.98,E2 -9255.98} C_VEL
LIN {X 0,Y 441.11,Z 482.641,A -85,B 0,C 180,E1 -9257.01,E2 -9257.01} C_VEL
LIN {X 0,Y 440.464,Z 491.818,A -85,B 0,C 180,E1 -9258.028,E2 -9258.028} C_VEL
LIN {X 0,Y 439.982,Z 500.317,A -85,B 0,C 180,E1 -9259.182,E2 -9259.182} C_VEL
LIN {X 0,Y 439.436,Z 508.573,A -85,B 0,C 180,E1 -9260.565,E2 -9260.565} C_VEL
LIN {X 0,Y 438.961,Z 515.225,A -85,B 0,C 180,E1 -9261.947,E2 -9261.947} C_VEL
LIN {X 0,Y 438.726,Z 519.558,A -85,B 0,C 180,E1 -9263.053,E2 -9263.053} C_VEL
LIN {X 0,Y 437.973,Z 521.988,A -85,B 0,C 180,E1 -9263.75,E2 -9263.75} C_VEL
LIN {X 0,Y 434.964,Z 525.389,A -85,B 0,C 180,E1 -9264.907,E2 -9264.907} C_VEL
LIN {X 0,Y 432.461,Z 527.595,A -85,B 0,C 180,E1 -9265.865,E2 -9265.865} C_VEL
LIN {X 0,Y 431.397,Z 528.959,A -85,B 0,C 180,E1 -9266.618,E2 -9266.618} C_VEL
LIN {X 0,Y 431.315,Z 529.317,A -85,B 0,C 180,E1 -9266.875,E2 -9266.875} C_VEL
LIN {X 0,Y 431.225,Z 530.799,A -85,B 0,C 180,E1 -9268.132,E2 -9268.132} C_VEL
LIN {X 0,Y 431.168,Z 531.648,A -85,B 0,C 180,E1 -9270,E2 -9270} C_VEL
LIN {X 0,Y 431.172,Z 531.46,A -85,B 0,C 180,E1 -9270.934,E2 -9270.934} C_VEL
LIN {X 0,Y 431.324,Z 529.908,A -85,B 0,C 180,E1 -9272.802,E2 -9272.802} C_VEL
LIN {X 0,Y 431.319,Z 528.555,A -85,B 0,C 180,E1 -9273.737,E2 -9273.737} C_VEL
LIN {X 0,Y 431.427,Z 525.691,A -85,B 0,C 180,E1 -9275.14,E2 -9275.14} C_VEL
LIN {X 0,Y 431.635,Z 521.407,A -85,B 0,C 180,E1 -9276.674,E2 -9276.674} C_VEL
LIN {X 0,Y 431.872,Z 516.795,A -85,B 0,C 180,E1 -9277.951,E2 -9277.951} C_VEL
LIN {X 0,Y 432.304,Z 510.485,A -85,B 0,C 180,E1 -9279.356,E2 -9279.356} C_VEL
LIN {X 0,Y 432.811,Z 502.586,A -85,B 0,C 180,E1 -9280.763,E2 -9280.763} C_VEL
LIN {X 0,Y 433.502,Z 492.757,A -85,B 0,C 180,E1 -9282.167,E2 -9282.167} C_VEL
LIN {X 0,Y 434.22,Z 483.113,A -85,B 0,C 180,E1 -9283.266,E2 -9283.266} C_VEL
LIN {X 0,Y 434.762,Z 472.226,A -85,B 0,C 180,E1 -9284.272,E2 -9284.272} C_VEL
LIN {X 0,Y 435.371,Z 461.045,A -85,B 0,C 180,E1 -9285.088,E2 -9285.088} C_VEL
LIN {X 0,Y 435.86,Z 448.464,A -85,B 0,C 180,E1 -9285.789,E2 -9285.789} C_VEL
LIN {X 0,Y 433.44,Z 435.731,A -85,B 0,C 180,E1 -9286.4,E2 -9286.4} C_VEL
LIN {X 0,Y 431.441,Z 427.348,A -85,B 0,C 180,E1 -9286.743,E2 -9286.743} C_VEL
LIN {X 0,Y 431.582,Z 423.712,A -85,B 0,C 180,E1 -9289.18,E2 -9289.18} C_VEL
LIN {X 0,Y 431.656,Z 418.274,A -85,B 0,C 180,E1 -9293.002,E2 -9293.002} C_VEL
LIN {X 0,Y 431.828,Z 414.07,A -85,B 0,C 180,E1 -9296.067,E2 -9296.067} C_VEL
LIN {X 0,Y 431.978,Z 409.859,A -85,B 0,C 180,E1 -9299.215,E2 -9299.215} C_VEL
LIN {X 0,Y 432.162,Z 405.634,A -85,B 0,C 180,E1 -9302.457,E2 -9302.457} C_VEL
LIN {X 0,Y 432.229,Z 402.787,A -85,B 0,C 180,E1 -9304.688,E2 -9304.688} C_VEL
LIN {X 0,Y 432.202,Z 401.652,A -85,B 0,C 180,E1 -9305.605,E2 -9305.605} C_VEL
LIN {X 0,Y 432.344,Z 401.633,A -85,B 0,C 180,E1 -9308.715,E2 -9308.715} C_VEL
LIN {X 0,Y 432.338,Z 401.63,A -85,B 0,C 180,E1 -9311.797,E2 -9311.797} C_VEL
LIN {X 0,Y 432.342,Z 401.632,A -85,B 0,C 180,E1 -9314.347,E2 -9314.347} C_VEL
LIN {X 0,Y 432.322,Z 401.635,A -85,B 0,C 180,E1 -9317.016,E2 -9317.016} C_VEL
LIN {X 0,Y 432.339,Z 401.628,A -85,B 0,C 180,E1 -9319.82,E2 -9319.82} C_VEL
LIN {X 0,Y 432.318,Z 401.633,A -85,B 0,C 180,E1 -9323.023,E2 -9323.023} C_VEL
LIN {X 0,Y 432.362,Z 401.629,A -85,B 0,C 180,E1 -9325.997,E2 -9325.997} C_VEL
LIN {X 0,Y 432.35,Z 401.628,A -85,B 0,C 180,E1 -9329.49,E2 -9329.49} C_VEL
LIN {X 0,Y 432.395,Z 401.623,A -85,B 0,C 180,E1 -9332.928,E2 -9332.928} C_VEL
LIN {X 0,Y 432.371,Z 401.628,A -85,B 0,C 180,E1 -9336.023,E2 -9336.023} C_VEL
LIN {X 0,Y 432.353,Z 401.628,A -85,B 0,C 180,E1 -9339.046,E2 -9339.046} C_VEL
LIN {X 0,Y 432.377,Z 401.627,A -85,B 0,C 180,E1 -9342.011,E2 -9342.011} C_VEL
LIN {X 0,Y 432.398,Z 401.622,A -85,B 0,C 180,E1 -9344.926,E2 -9344.926} C_VEL
LIN {X 0,Y 432.463,Z 401.616,A -85,B 0,C 180,E1 -9347.803,E2 -9347.803} C_VEL
LIN {X 0,Y 432.495,Z 401.612,A -85,B 0,C 180,E1 -9351.59,E2 -9351.59} C_VEL
LIN {X 0,Y 432.6,Z 401.599,A -85,B 0,C 180,E1 -9354.406,E2 -9354.406} C_VEL
LIN {X 0,Y 432.607,Z 401.6,A -85,B 0,C 180,E1 -9358.138,E2 -9358.138} C_VEL
LIN {X 0,Y 432.735,Z 401.584,A -85,B 0,C 180,E1 -9360,E2 -9360} C_VEL
LIN {X 0,Y 432.595,Z 401.596,A -85,B 0,C 180,E1 -9362.794,E2 -9362.794} C_VEL
LIN {X 0,Y 432.576,Z 401.6,A -85,B 0,C 180,E1 -9366.53,E2 -9366.53} C_VEL
LIN {X 0,Y 432.448,Z 401.619,A -85,B 0,C 180,E1 -9369.353,E2 -9369.353} C_VEL
LIN {X 0,Y 432.448,Z 401.616,A -85,B 0,C 180,E1 -9372.812,E2 -9372.812} C_VEL
LIN {X 0,Y 432.416,Z 401.619,A -85,B 0,C 180,E1 -9376.479,E2 -9376.479} C_VEL
LIN {X 0,Y 432.342,Z 401.631,A -85,B 0,C 180,E1 -9379.96,E2 -9379.96} C_VEL
LIN {X 0,Y 432.32,Z 401.635,A -85,B 0,C 180,E1 -9382.964,E2 -9382.964} C_VEL
LIN {X 0,Y 432.364,Z 401.626,A -85,B 0,C 180,E1 -9386.033,E2 -9386.033} C_VEL
LIN {X 0,Y 432.346,Z 401.634,A -85,B 0,C 180,E1 -9389.187,E2 -9389.187} C_VEL
LIN {X 0,Y 432.326,Z 401.632,A -85,B 0,C 180,E1 -9392.443,E2 -9392.443} C_VEL
LIN {X 0,Y 432.348,Z 401.63,A -85,B 0,C 180,E1 -9395.632,E2 -9395.632} C_VEL
LIN {X 0,Y 432.353,Z 401.629,A -85,B 0,C 180,E1 -9398.716,E2 -9398.716} C_VEL
LIN {X 0,Y 432.336,Z 401.628,A -85,B 0,C 180,E1 -9401.797,E2 -9401.797} C_VEL
LIN {X 0,Y 432.336,Z 401.635,A -85,B 0,C 180,E1 -9404.347,E2 -9404.347} C_VEL
LIN {X 0,Y 432.327,Z 401.633,A -85,B 0,C 180,E1 -9407.015,E2 -9407.015} C_VEL
LIN {X 0,Y 432.4,Z 401.761,A -85,B 0,C 180,E1 -9409.891,E2 -9409.891} C_VEL
LIN {X 0,Y 433.306,Z 407.455,A -85,B 0,C 180,E1 -9413.121,E2 -9413.121} C_VEL
LIN {X 0,Y 433.477,Z 411.833,A -85,B 0,C 180,E1 -9415.427,E2 -9415.427} C_VEL
LIN {X 0,Y 433.037,Z 418.393,A -85,B 0,C 180,E1 -9418.711,E2 -9418.711} C_VEL
LIN {X 0,Y 432.781,Z 423.673,A -85,B 0,C 180,E1 -9421.273,E2 -9421.273} C_VEL
LIN {X 0,Y 432.346,Z 431.591,A -85,B 0,C 180,E1 -9424.998,E2 -9424.998} C_VEL
LIN {X 0,Y 432.022,Z 439.258,A -85,B 0,C 180,E1 -9428.529,E2 -9428.529} C_VEL
LIN {X 0,Y 431.742,Z 445.774,A -85,B 0,C 180,E1 -9431.493,E2 -9431.493} C_VEL
LIN {X 0,Y 431.661,Z 449.89,A -85,B 0,C 180,E1 -9433.309,E2 -9433.309} C_VEL
LIN {X 0,Y 433.888,Z 462.697,A -85,B 0,C 180,E1 -9433.764,E2 -9433.764} C_VEL
LIN {X 0,Y 435.536,Z 475.228,A -85,B 0,C 180,E1 -9434.379,E2 -9434.379} C_VEL
LIN {X 0,Y 434.874,Z 488.072,A -85,B 0,C 180,E1 -9435.134,E2 -9435.134} C_VEL
LIN {X 0,Y 434.237,Z 498.749,A -85,B 0,C 180,E1 -9435.95,E2 -9435.95} C_VEL
LIN {X 0,Y 433.565,Z 509.657,A -85,B 0,C 180,E1 -9437.002,E2 -9437.002} C_VEL
LIN {X 0,Y 433.019,Z 518.556,A -85,B 0,C 180,E1 -9438.057,E2 -9438.057} C_VEL
LIN {X 0,Y 432.307,Z 528.222,A -85,B 0,C 180,E1 -9439.462,E2 -9439.462} C_VEL
LIN {X 0,Y 431.879,Z 535.921,A -85,B 0,C 180,E1 -9440.871,E2 -9440.871} C_VEL
LIN {X 0,Y 431.536,Z 543.02,A -85,B 0,C 180,E1 -9442.514,E2 -9442.514} C_VEL
LIN {X 0,Y 431.292,Z 548.018,A -85,B 0,C 180,E1 -9444.01,E2 -9444.01} C_VEL
LIN {X 0,Y 431.275,Z 551.354,A -85,B 0,C 180,E1 -9445.326,E2 -9445.326} C_VEL
LIN {X 0,Y 431.189,Z 553.215,A -85,B 0,C 180,E1 -9446.262,E2 -9446.262} C_VEL
LIN {X 0,Y 431.236,Z 554.613,A -85,B 0,C 180,E1 -9447.197,E2 -9447.197} C_VEL
LIN {X 0,Y 431.203,Z 555.609,A -85,B 0,C 180,E1 -9448.132,E2 -9448.132} C_VEL
LIN {X 0,Y 431.167,Z 556.433,A -85,B 0,C 180,E1 -9450,E2 -9450} C_VEL
LIN {X 0,Y 431.203,Z 555.609,A -85,B 0,C 180,E1 -9451.868,E2 -9451.868} C_VEL
LIN {X 0,Y 431.236,Z 554.614,A -85,B 0,C 180,E1 -9452.802,E2 -9452.802} C_VEL
LIN {X 0,Y 431.189,Z 553.215,A -85,B 0,C 180,E1 -9453.738,E2 -9453.738} C_VEL
LIN {X 0,Y 431.301,Z 550.279,A -85,B 0,C 180,E1 -9455.142,E2 -9455.142} C_VEL
LIN {X 0,Y 431.378,Z 546.301,A -85,B 0,C 180,E1 -9456.548,E2 -9456.548} C_VEL
LIN {X 0,Y 431.68,Z 540.189,A -85,B 0,C 180,E1 -9458.19,E2 -9458.19} C_VEL
LIN {X 0,Y 432.01,Z 533.509,A -85,B 0,C 180,E1 -9459.599,E2 -9459.599} C_VEL
LIN {X 0,Y 432.532,Z 525.224,A -85,B 0,C 180,E1 -9461.006,E2 -9461.006} C_VEL
LIN {X 0,Y 433.157,Z 516.735,A -85,B 0,C 180,E1 -9462.177,E2 -9462.177} C_VEL
LIN {X 0,Y 433.77,Z 507.016,A -85,B 0,C 180,E1 -9463.271,E2 -9463.271} C_VEL
LIN {X 0,Y 434.409,Z 495.864,A -85,B 0,C 180,E1 -9464.283,E2 -9464.283} C_VEL
LIN {X 0,Y 435.051,Z 484.486,A -85,B 0,C 180,E1 -9465.099,E2 -9465.099} C_VEL
LIN {X 0,Y 435.423,Z 474.022,A -85,B 0,C 180,E1 -9465.685,E2 -9465.685} C_VEL
LIN {X 0,Y 433.601,Z 460.832,A -85,B 0,C 180,E1 -9466.306,E2 -9466.306} C_VEL
LIN {X 0,Y 431.67,Z 449.715,A -85,B 0,C 180,E1 -9466.705,E2 -9466.705} C_VEL
LIN {X 0,Y 431.92,Z 441.422,A -85,B 0,C 180,E1 -9470.477,E2 -9470.477} C_VEL
LIN {X 0,Y 432.151,Z 434.879,A -85,B 0,C 180,E1 -9473.481,E2 -9473.481} C_VEL
LIN {X 0,Y 432.485,Z 428.032,A -85,B 0,C 180,E1 -9476.649,E2 -9476.649} C_VEL
LIN {X 0,Y 432.898,Z 421.654,A -85,B 0,C 180,E1 -9479.68,E2 -9479.68} C_VEL
LIN {X 0,Y 433.174,Z 415.982,A -85,B 0,C 180,E1 -9482.47,E2 -9482.47} C_VEL
LIN {X 0,Y 433.496,Z 410.73,A -85,B 0,C 180,E1 -9485.137,E2 -9485.137} C_VEL
LIN {X 0,Y 433.178,Z 406.608,A -85,B 0,C 180,E1 -9487.345,E2 -9487.345} C_VEL
LIN {X 0,Y 432.385,Z 401.628,A -85,B 0,C 180,E1 -9490.187,E2 -9490.187} C_VEL
LIN {X 0,Y 432.325,Z 401.634,A -85,B 0,C 180,E1 -9493.06,E2 -9493.06} C_VEL
LIN {X 0,Y 432.334,Z 401.635,A -85,B 0,C 180,E1 -9495.665,E2 -9495.665} C_VEL
LIN {X 0,Y 432.334,Z 401.629,A -85,B 0,C 180,E1 -9498.398,E2 -9498.398} C_VEL
LIN {X 0,Y 432.348,Z 401.628,A -85,B 0,C 180,E1 -9501.851,E2 -9501.851} C_VEL
LIN {X 0,Y 432.342,Z 401.632,A -85,B 0,C 180,E1 -9505.323,E2 -9505.323} C_VEL
LIN {X 0,Y 432.323,Z 401.634,A -85,B 0,C 180,E1 -9508.654,E2 -9508.654} C_VEL
LIN {X 0,Y 432.384,Z 401.622,A -85,B 0,C 180,E1 -9511.877,E2 -9511.877} C_VEL
LIN {X 0,Y 432.347,Z 401.63,A -85,B 0,C 180,E1 -9514.998,E2 -9514.998} C_VEL
LIN {X 0,Y 432.359,Z 401.629,A -85,B 0,C 180,E1 -9518.046,E2 -9518.046} C_VEL
LIN {X 0,Y 432.389,Z 401.626,A -85,B 0,C 180,E1 -9521.03,E2 -9521.03} C_VEL
LIN {X 0,Y 432.433,Z 401.618,A -85,B 0,C 180,E1 -9523.961,E2 -9523.961} C_VEL
LIN {X 0,Y 432.483,Z 401.612,A -85,B 0,C 180,E1 -9527.804,E2 -9527.804} C_VEL
LIN {X 0,Y 432.494,Z 401.611,A -85,B 0,C 180,E1 -9531.59,E2 -9531.59} C_VEL
LIN {X 0,Y 432.599,Z 401.6,A -85,B 0,C 180,E1 -9534.406,E2 -9534.406} C_VEL
LIN {X 0,Y 432.606,Z 401.6,A -85,B 0,C 180,E1 -9538.138,E2 -9538.138} C_VEL
LIN {X 0,Y 432.736,Z 401.583,A -85,B 0,C 180,E1 -9540,E2 -9540} C_VEL
LIN {X 0,Y 432.593,Z 401.599,A -85,B 0,C 180,E1 -9542.794,E2 -9542.794} C_VEL
LIN {X 0,Y 432.575,Z 401.603,A -85,B 0,C 180,E1 -9546.53,E2 -9546.53} C_VEL
LIN {X 0,Y 432.447,Z 401.616,A -85,B 0,C 180,E1 -9549.353,E2 -9549.353} C_VEL
LIN {X 0,Y 432.447,Z 401.615,A -85,B 0,C 180,E1 -9552.812,E2 -9552.812} C_VEL
LIN {X 0,Y 432.414,Z 401.622,A -85,B 0,C 180,E1 -9556.479,E2 -9556.479} C_VEL
LIN {X 0,Y 432.341,Z 401.632,A -85,B 0,C 180,E1 -9559.96,E2 -9559.96} C_VEL
LIN {X 0,Y 432.32,Z 401.632,A -85,B 0,C 180,E1 -9562.964,E2 -9562.964} C_VEL
LIN {X 0,Y 432.363,Z 401.628,A -85,B 0,C 180,E1 -9566.033,E2 -9566.033} C_VEL
LIN {X 0,Y 432.345,Z 401.631,A -85,B 0,C 180,E1 -9569.187,E2 -9569.187} C_VEL
LIN {X 0,Y 432.325,Z 401.632,A -85,B 0,C 180,E1 -9572.443,E2 -9572.443} C_VEL
LIN {X 0,Y 432.348,Z 401.632,A -85,B 0,C 180,E1 -9575.632,E2 -9575.632} C_VEL
LIN {X 0,Y 432.355,Z 401.626,A -85,B 0,C 180,E1 -9578.717,E2 -9578.717} C_VEL
LIN {X 0,Y 432.335,Z 401.631,A -85,B 0,C 180,E1 -9581.797,E2 -9581.797} C_VEL
LIN {X 0,Y 432.335,Z 401.63,A -85,B 0,C 180,E1 -9584.347,E2 -9584.347} C_VEL
LIN {X 0,Y 432.327,Z 401.634,A -85,B 0,C 180,E1 -9587.015,E2 -9587.015} C_VEL
LIN {X 0,Y 432.335,Z 401.631,A -85,B 0,C 180,E1 -9589.821,E2 -9589.821} C_VEL
LIN {X 0,Y 432.293,Z 401.638,A -85,B 0,C 180,E1 -9593.021,E2 -9593.021} C_VEL
LIN {X 0,Y 432.198,Z 401.651,A -85,B 0,C 180,E1 -9594.396,E2 -9594.396} C_VEL
LIN {X 0,Y 432.208,Z 404.076,A -85,B 0,C 180,E1 -9596.436,E2 -9596.436} C_VEL
LIN {X 0,Y 432.081,Z 408.308,A -85,B 0,C 180,E1 -9599.72,E2 -9599.72} C_VEL
LIN {X 0,Y 431.849,Z 412.521,A -85,B 0,C 180,E1 -9602.892,E2 -9602.892} C_VEL
LIN {X 0,Y 431.744,Z 416.714,A -85,B 0,C 180,E1 -9605.986,E2 -9605.986} C_VEL
LIN {X 0,Y 431.565,Z 420.982,A -85,B 0,C 180,E1 -9609.006,E2 -9609.006} C_VEL
LIN {X 0,Y 431.508,Z 425.284,A -85,B 0,C 180,E1 -9611.974,E2 -9611.974} C_VEL
LIN {X 0,Y 431.515,Z 427.357,A -85,B 0,C 180,E1 -9613.362,E2 -9613.362} C_VEL
LIN {X 0,Y 434.792,Z 442.183,A -85,B 0,C 180,E1 -9613.984,E2 -9613.984} C_VEL
LIN {X 0,Y 435.882,Z 449.022,A -85,B 0,C 180,E1 -9614.332,E2 -9614.332} C_VEL
LIN {X 0,Y 435.352,Z 461.432,A -85,B 0,C 180,E1 -9615.031,E2 -9615.031} C_VEL
LIN {X 0,Y 434.703,Z 473.673,A -85,B 0,C 180,E1 -9615.941,E2 -9615.941} C_VEL
LIN {X 0,Y 434.058,Z 484.931,A -85,B 0,C 180,E1 -9617.017,E2 -9617.017} C_VEL
LIN {X 0,Y 433.412,Z 493.837,A -85,B 0,C 180,E1 -9618.068,E2 -9618.068} C_VEL
LIN {X 0,Y 432.754,Z 503.483,A -85,B 0,C 180,E1 -9619.473,E2 -9619.473} C_VEL
LIN {X 0,Y 432.246,Z 511.178,A -85,B 0,C 180,E1 -9620.879,E2 -9620.879} C_VEL
LIN {X 0,Y 431.735,Z 518.24,A -85,B 0,C 180,E1 -9622.517,E2 -9622.517} C_VEL
LIN {X 0,Y 431.622,Z 522.938,A -85,B 0,C 180,E1 -9623.925,E2 -9623.925} C_VEL
LIN {X 0,Y 431.352,Z 526.541,A -85,B 0,C 180,E1 -9625.327,E2 -9625.327} C_VEL
LIN {X 0,Y 431.315,Z 529.317,A -85,B 0,C 180,E1 -9626.875,E2 -9626.875} C_VEL
LIN {X 0,Y 430.641,Z 530.372,A -85,B 0,C 180,E1 -9627.643,E2 -9627.643} C_VEL
LIN {X 0,Y 427.712,Z 531.578,A -85,B 0,C 180,E1 -9628.899,E2 -9628.899} C_VEL
LIN {X 0,Y 425.234,Z 531.938,A -85,B 0,C 180,E1 -9629.918,E2 -9629.918} C_VEL
LIN {X 0,Y 424.174,Z 531.789,A -85,B 0,C 180,E1 -9630.706,E2 -9630.706} C_VEL
LIN {X 0,Y 424.092,Z 531.649,A -85,B 0,C 180,E1 -9630.973,E2 -9630.973} C_VEL
LIN {X 0,Y 424.238,Z 530.111,A -85,B 0,C 180,E1 -9632.849,E2 -9632.849} C_VEL
LIN {X 0,Y 424.225,Z 528.758,A -85,B 0,C 180,E1 -9633.8,E2 -9633.8} C_VEL
LIN {X 0,Y 424.376,Z 525.893,A -85,B 0,C 180,E1 -9635.226,E2 -9635.226} C_VEL
LIN {X 0,Y 424.563,Z 521.938,A -85,B 0,C 180,E1 -9636.678,E2 -9636.678} C_VEL
LIN {X 0,Y 424.819,Z 516.998,A -85,B 0,C 180,E1 -9638.084,E2 -9638.084} C_VEL
LIN {X 0,Y 425.305,Z 510.687,A -85,B 0,C 180,E1 -9639.512,E2 -9639.512} C_VEL
LIN {X 0,Y 425.834,Z 502.787,A -85,B 0,C 180,E1 -9640.941,E2 -9640.941} C_VEL
LIN {X 0,Y 426.41,Z 494.733,A -85,B 0,C 180,E1 -9642.131,E2 -9642.131} C_VEL
LIN {X 0,Y 427.211,Z 484.899,A -85,B 0,C 180,E1 -9643.316,E2 -9643.316} C_VEL
LIN {X 0,Y 427.683,Z 475.23,A -85,B 0,C 180,E1 -9644.27,E2 -9644.27} C_VEL
LIN {X 0,Y 428.352,Z 464.762,A -85,B 0,C 180,E1 -9645.098,E2 -9645.098} C_VEL
LIN {X 0,Y 428.948,Z 452.154,A -85,B 0,C 180,E1 -9645.868,E2 -9645.868} C_VEL
LIN {X 0,Y 428.91,Z 448.661,A -85,B 0,C 180,E1 -9646.052,E2 -9646.052} C_VEL
LIN {X 0,Y 426.574,Z 436.819,A -85,B 0,C 180,E1 -9646.642,E2 -9646.642} C_VEL
LIN {X 0,Y 424.357,Z 427.552,A -85,B 0,C 180,E1 -9647.024,E2 -9647.024} C_VEL
LIN {X 0,Y 424.503,Z 424.148,A -85,B 0,C 180,E1 -9649.337,E2 -9649.337} C_VEL
LIN {X 0,Y 424.556,Z 419.871,A -85,B 0,C 180,E1 -9652.379,E2 -9652.379} C_VEL
LIN {X 0,Y 424.726,Z 415.615,A -85,B 0,C 180,E1 -9655.482,E2 -9655.482} C_VEL
LIN {X 0,Y 424.901,Z 411.295,A -85,B 0,C 180,E1 -9658.76,E2 -9658.76} C_VEL
LIN {X 0,Y 425.075,Z 407.172,A -85,B 0,C 180,E1 -9661.943,E2 -9661.943} C_VEL
LIN {X 0,Y 425.194,Z 404.237,A -85,B 0,C 180,E1 -9664.264,E2 -9664.264} C_VEL
LIN {X 0,Y 425.177,Z 402.901,A -85,B 0,C 180,E1 -9665.348,E2 -9665.348} C_VEL
LIN {X 0,Y 425.215,Z 402.521,A -85,B 0,C 180,E1 -9666.514,E2 -9666.514} C_VEL
LIN {X 0,Y 425.295,Z 402.509,A -85,B 0,C 180,E1 -9669.043,E2 -9669.043} C_VEL
LIN {X 0,Y 425.281,Z 402.512,A -85,B 0,C 180,E1 -9672.653,E2 -9672.653} C_VEL
LIN {X 0,Y 425.264,Z 402.512,A -85,B 0,C 180,E1 -9676.044,E2 -9676.044} C_VEL
LIN {X 0,Y 425.277,Z 402.513,A -85,B 0,C 180,E1 -9678.621,E2 -9678.621} C_VEL
LIN {X 0,Y 425.316,Z 402.504,A -85,B 0,C 180,E1 -9681.103,E2 -9681.103} C_VEL
LIN {X 0,Y 425.302,Z 402.509,A -85,B 0,C 180,E1 -9684.664,E2 -9684.664} C_VEL
LIN {X 0,Y 425.268,Z 402.513,A -85,B 0,C 180,E1 -9688.073,E2 -9688.073} C_VEL
LIN {X 0,Y 425.334,Z 402.501,A -85,B 0,C 180,E1 -9691.368,E2 -9691.368} C_VEL
LIN {X 0,Y 425.357,Z 402.498,A -85,B 0,C 180,E1 -9693.505,E2 -9693.505} C_VEL
LIN {X 0,Y 425.308,Z 402.507,A -85,B 0,C 180,E1 -9696.635,E2 -9696.635} C_VEL
LIN {X 0,Y 425.331,Z 402.505,A -85,B 0,C 180,E1 -9700.364,E2 -9700.364} C_VEL
LIN {X 0,Y 425.391,Z 402.497,A -85,B 0,C 180,E1 -9703.688,E2 -9703.688} C_VEL
LIN {X 0,Y 425.415,Z 402.492,A -85,B 0,C 180,E1 -9707.598,E2 -9707.598} C_VEL
LIN {X 0,Y 425.446,Z 402.489,A -85,B 0,C 180,E1 -9711.45,E2 -9711.45} C_VEL
LIN {X 0,Y 425.557,Z 402.477,A -85,B 0,C 180,E1 -9714.313,E2 -9714.313} C_VEL
LIN {X 0,Y 425.576,Z 402.476,A -85,B 0,C 180,E1 -9718.107,E2 -9718.107} C_VEL
LIN {X 0,Y 425.705,Z 402.46,A -85,B 0,C 180,E1 -9720,E2 -9720} C_VEL
LIN {X 0,Y 425.549,Z 402.474,A -85,B 0,C 180,E1 -9722.84,E2 -9722.84} C_VEL
LIN {X 0,Y 425.534,Z 402.477,A -85,B 0,C 180,E1 -9726.639,E2 -9726.639} C_VEL
LIN {X 0,Y 425.406,Z 402.496,A -85,B 0,C 180,E1 -9729.509,E2 -9729.509} C_VEL
LIN {X 0,Y 425.407,Z 402.493,A -85,B 0,C 180,E1 -9732.91,E2 -9732.91} C_VEL
LIN {X 0,Y 425.365,Z 402.497,A -85,B 0,C 180,E1 -9736.605,E2 -9736.605} C_VEL
LIN {X 0,Y 425.332,Z 402.505,A -85,B 0,C 180,E1 -9739.636,E2 -9739.636} C_VEL
LIN {X 0,Y 425.308,Z 402.508,A -85,B 0,C 180,E1 -9743.365,E2 -9743.365} C_VEL
LIN {X 0,Y 425.35,Z 402.501,A -85,B 0,C 180,E1 -9746.844,E2 -9746.844} C_VEL
LIN {X 0,Y 425.294,Z 402.508,A -85,B 0,C 180,E1 -9749.719,E2 -9749.719} C_VEL
LIN {X 0,Y 425.285,Z 402.512,A -85,B 0,C 180,E1 -9753.048,E2 -9753.048} C_VEL
LIN {X 0,Y 425.287,Z 402.508,A -85,B 0,C 180,E1 -9755.929,E2 -9755.929} C_VEL
LIN {X 0,Y 425.303,Z 402.509,A -85,B 0,C 180,E1 -9759.044,E2 -9759.044} C_VEL
LIN {X 0,Y 425.277,Z 402.511,A -85,B 0,C 180,E1 -9762.653,E2 -9762.653} C_VEL
LIN {X 0,Y 425.271,Z 402.512,A -85,B 0,C 180,E1 -9766.045,E2 -9766.045} C_VEL
LIN {X 0,Y 425.345,Z 402.607,A -85,B 0,C 180,E1 -9769.618,E2 -9769.618} C_VEL
LIN {X 0,Y 426.139,Z 407.372,A -85,B 0,C 180,E1 -9772.395,E2 -9772.395} C_VEL
LIN {X 0,Y 426.499,Z 411.722,A -85,B 0,C 180,E1 -9774.778,E2 -9774.778} C_VEL
LIN {X 0,Y 426.095,Z 418.269,A -85,B 0,C 180,E1 -9778.142,E2 -9778.142} C_VEL
LIN {X 0,Y 425.756,Z 424.093,A -85,B 0,C 180,E1 -9781.031,E2 -9781.031} C_VEL
LIN {X 0,Y 425.315,Z 431.437,A -85,B 0,C 180,E1 -9784.556,E2 -9784.556} C_VEL
LIN {X 0,Y 425.017,Z 438.37,A -85,B 0,C 180,E1 -9787.821,E2 -9787.821} C_VEL
LIN {X 0,Y 424.693,Z 445.585,A -85,B 0,C 180,E1 -9791.174,E2 -9791.174} C_VEL
LIN {X 0,Y 424.585,Z 449.546,A -85,B 0,C 180,E1 -9793.017,E2 -9793.017} C_VEL
LIN {X 0,Y 426.955,Z 462.992,A -85,B 0,C 180,E1 -9793.512,E2 -9793.512} C_VEL
LIN {X 0,Y 428.623,Z 476.16,A -85,B 0,C 180,E1 -9794.181,E2 -9794.181} C_VEL
LIN {X 0,Y 428.011,Z 487.872,A -85,B 0,C 180,E1 -9794.89,E2 -9794.89} C_VEL
LIN {X 0,Y 427.35,Z 498.549,A -85,B 0,C 180,E1 -9795.719,E2 -9795.719} C_VEL
LIN {X 0,Y 426.619,Z 509.455,A -85,B 0,C 180,E1 -9796.787,E2 -9796.787} C_VEL
LIN {X 0,Y 426.056,Z 518.353,A -85,B 0,C 180,E1 -9797.859,E2 -9797.859} C_VEL
LIN {X 0,Y 425.298,Z 528.019,A -85,B 0,C 180,E1 -9799.286,E2 -9799.286} C_VEL
LIN {X 0,Y 424.834,Z 535.717,A -85,B 0,C 180,E1 -9800.718,E2 -9800.718} C_VEL
LIN {X 0,Y 424.453,Z 542.816,A -85,B 0,C 180,E1 -9802.388,E2 -9802.388} C_VEL
LIN {X 0,Y 424.247,Z 547.17,A -85,B 0,C 180,E1 -9803.695,E2 -9803.695} C_VEL
LIN {X 0,Y 424.204,Z 551.151,A -85,B 0,C 180,E1 -9805.248,E2 -9805.248} C_VEL
LIN {X 0,Y 424.101,Z 553.011,A -85,B 0,C 180,E1 -9806.199,E2 -9806.199} C_VEL
LIN {X 0,Y 424.132,Z 554.409,A -85,B 0,C 180,E1 -9807.15,E2 -9807.15} C_VEL
LIN {X 0,Y 424.129,Z 555.406,A -85,B 0,C 180,E1 -9808.101,E2 -9808.101} C_VEL
LIN {X 0,Y 424.084,Z 556.229,A -85,B 0,C 180,E1 -9810,E2 -9810} C_VEL
LIN {X 0,Y 424.129,Z 555.405,A -85,B 0,C 180,E1 -9811.899,E2 -9811.899} C_VEL
LIN {X 0,Y 424.132,Z 554.409,A -85,B 0,C 180,E1 -9812.849,E2 -9812.849} C_VEL
LIN {X 0,Y 424.101,Z 553.01,A -85,B 0,C 180,E1 -9813.801,E2 -9813.801} C_VEL
LIN {X 0,Y 424.214,Z 550.074,A -85,B 0,C 180,E1 -9815.228,E2 -9815.228} C_VEL
LIN {X 0,Y 424.302,Z 546.096,A -85,B 0,C 180,E1 -9816.658,E2 -9816.658} C_VEL
LIN {X 0,Y 424.614,Z 539.983,A -85,B 0,C 180,E1 -9818.327,E2 -9818.327} C_VEL
LIN {X 0,Y 424.964,Z 533.302,A -85,B 0,C 180,E1 -9819.759,E2 -9819.759} C_VEL
LIN {X 0,Y 425.517,Z 525.017,A -85,B 0,C 180,E1 -9821.19,E2 -9821.19} C_VEL
LIN {X 0,Y 426.188,Z 516.528,A -85,B 0,C 180,E1 -9822.379,E2 -9822.379} C_VEL
LIN {X 0,Y 426.9,Z 506.067,A -85,B 0,C 180,E1 -9823.565,E2 -9823.565} C_VEL
LIN {X 0,Y 427.507,Z 495.655,A -85,B 0,C 180,E1 -9824.519,E2 -9824.519} C_VEL
LIN {X 0,Y 428.193,Z 484.278,A -85,B 0,C 180,E1 -9825.347,E2 -9825.347} C_VEL
LIN {X 0,Y 428.532,Z 474.944,A -85,B 0,C 180,E1 -9825.883,E2 -9825.883} C_VEL
LIN {X 0,Y 426.775,Z 461.938,A -85,B 0,C 180,E1 -9826.53,E2 -9826.53} C_VEL
LIN {X 0,Y 424.59,Z 449.507,A -85,B 0,C 180,E1 -9826.996,E2 -9826.996} C_VEL
LIN {X 0,Y 424.891,Z 441.244,A -85,B 0,C 180,E1 -9830.832,E2 -9830.832} C_VEL
LIN {X 0,Y 425.139,Z 434.716,A -85,B 0,C 180,E1 -9833.892,E2 -9833.892} C_VEL
LIN {X 0,Y 425.441,Z 428.422,A -85,B 0,C 180,E1 -9836.868,E2 -9836.868} C_VEL
LIN {X 0,Y 425.862,Z 422.606,A -85,B 0,C 180,E1 -9839.676,E2 -9839.676} C_VEL
LIN {X 0,Y 426.212,Z 416.058,A -85,B 0,C 180,E1 -9842.967,E2 -9842.967} C_VEL
LIN {X 0,Y 426.493,Z 411.707,A -85,B 0,C 180,E1 -9845.222,E2 -9845.222} C_VEL
LIN {X 0,Y 426.121,Z 407.26,A -85,B 0,C 180,E1 -9847.659,E2 -9847.659} C_VEL
LIN {X 0,Y 425.348,Z 402.574,A -85,B 0,C 180,E1 -9850.382,E2 -9850.382} C_VEL
LIN {X 0,Y 425.27,Z 402.514,A -85,B 0,C 180,E1 -9853.955,E2 -9853.955} C_VEL
LIN {X 0,Y 425.276,Z 402.511,A -85,B 0,C 180,E1 -9857.347,E2 -9857.347} C_VEL
LIN {X 0,Y 425.302,Z 402.51,A -85,B 0,C 180,E1 -9860.956,E2 -9860.956} C_VEL
LIN {X 0,Y 425.302,Z 402.509,A -85,B 0,C 180,E1 -9864.664,E2 -9864.664} C_VEL
LIN {X 0,Y 425.266,Z 402.511,A -85,B 0,C 180,E1 -9868.073,E2 -9868.073} C_VEL
LIN {X 0,Y 425.333,Z 402.502,A -85,B 0,C 180,E1 -9871.368,E2 -9871.368} C_VEL
LIN {X 0,Y 425.355,Z 402.499,A -85,B 0,C 180,E1 -9873.505,E2 -9873.505} C_VEL
LIN {X 0,Y 425.306,Z 402.509,A -85,B 0,C 180,E1 -9876.635,E2 -9876.635} C_VEL
LIN {X 0,Y 425.33,Z 402.505,A -85,B 0,C 180,E1 -9880.364,E2 -9880.364} C_VEL
LIN {X 0,Y 425.39,Z 402.494,A -85,B 0,C 180,E1 -9883.688,E2 -9883.688} C_VEL
LIN {X 0,Y 425.432,Z 402.489,A -85,B 0,C 180,E1 -9887.599,E2 -9887.599} C_VEL
LIN {X 0,Y 425.445,Z 402.488,A -85,B 0,C 180,E1 -9891.45,E2 -9891.45} C_VEL
LIN {X 0,Y 425.556,Z 402.477,A -85,B 0,C 180,E1 -9894.313,E2 -9894.313} C_VEL
LIN {X 0,Y 425.575,Z 402.475,A -85,B 0,C 180,E1 -9898.107,E2 -9898.107} C_VEL
LIN {X 0,Y 425.706,Z 402.459,A -85,B 0,C 180,E1 -9900,E2 -9900} C_VEL
LIN {X 0,Y 425.547,Z 402.476,A -85,B 0,C 180,E1 -9902.84,E2 -9902.84} C_VEL
LIN {X 0,Y 425.533,Z 402.479,A -85,B 0,C 180,E1 -9906.646,E2 -9906.646} C_VEL
LIN {X 0,Y 425.405,Z 402.494,A -85,B 0,C 180,E1 -9909.509,E2 -9909.509} C_VEL
LIN {X 0,Y 425.406,Z 402.492,A -85,B 0,C 180,E1 -9912.91,E2 -9912.91} C_VEL
LIN {X 0,Y 425.363,Z 402.499,A -85,B 0,C 180,E1 -9916.605,E2 -9916.605} C_VEL
LIN {X 0,Y 425.33,Z 402.505,A -85,B 0,C 180,E1 -9919.636,E2 -9919.636} C_VEL
LIN {X 0,Y 425.307,Z 402.507,A -85,B 0,C 180,E1 -9923.365,E2 -9923.365} C_VEL
LIN {X 0,Y 425.349,Z 402.499,A -85,B 0,C 180,E1 -9926.844,E2 -9926.844} C_VEL
LIN {X 0,Y 425.293,Z 402.51,A -85,B 0,C 180,E1 -9929.72,E2 -9929.72} C_VEL
LIN {X 0,Y 425.284,Z 402.51,A -85,B 0,C 180,E1 -9933.048,E2 -9933.048} C_VEL
LIN {X 0,Y 425.287,Z 402.51,A -85,B 0,C 180,E1 -9935.929,E2 -9935.929} C_VEL
LIN {X 0,Y 425.305,Z 402.506,A -85,B 0,C 180,E1 -9939.045,E2 -9939.045} C_VEL
LIN {X 0,Y 425.277,Z 402.509,A -85,B 0,C 180,E1 -9942.653,E2 -9942.653} C_VEL
LIN {X 0,Y 425.27,Z 402.511,A -85,B 0,C 180,E1 -9946.045,E2 -9946.045} C_VEL
LIN {X 0,Y 425.277,Z 402.51,A -85,B 0,C 180,E1 -9948.622,E2 -9948.622} C_VEL
LIN {X 0,Y 425.307,Z 402.508,A -85,B 0,C 180,E1 -9951.102,E2 -9951.102} C_VEL
LIN {X 0,Y 425.187,Z 402.523,A -85,B 0,C 180,E1 -9954.089,E2 -9954.089} C_VEL
LIN {X 0,Y 425.141,Z 402.774,A -85,B 0,C 180,E1 -9954.649,E2 -9954.649} C_VEL
LIN {X 0,Y 425.114,Z 406.295,A -85,B 0,C 180,E1 -9957.473,E2 -9957.473} C_VEL
LIN {X 0,Y 424.958,Z 409.865,A -85,B 0,C 180,E1 -9960.255,E2 -9960.255} C_VEL
LIN {X 0,Y 424.801,Z 414.077,A -85,B 0,C 180,E1 -9963.468,E2 -9963.468} C_VEL
LIN {X 0,Y 424.611,Z 418.301,A -85,B 0,C 180,E1 -9966.594,E2 -9966.594} C_VEL
LIN {X 0,Y 424.484,Z 422.582,A -85,B 0,C 180,E1 -9969.654,E2 -9969.654} C_VEL
LIN {X 0,Y 424.432,Z 427.431,A -85,B 0,C 180,E1 -9972.994,E2 -9972.994} C_VEL
LIN {X 0,Y 424.45,Z 427.695,A -85,B 0,C 180,E1 -9973.095,E2 -9973.095} C_VEL
LIN {X 0,Y 427.517,Z 441.053,A -85,B 0,C 180,E1 -9973.65,E2 -9973.65} C_VEL
LIN {X 0,Y 429.01,Z 450.406,A -85,B 0,C 180,E1 -9974.135,E2 -9974.135} C_VEL
LIN {X 0,Y 428.438,Z 463.404,A -85,B 0,C 180,E1 -9974.906,E2 -9974.906} C_VEL
LIN {X 0,Y 427.787,Z 474.547,A -85,B 0,C 180,E1 -9975.766,E2 -9975.766} C_VEL
LIN {X 0,Y 427.143,Z 485.139,A -85,B 0,C 180,E1 -9976.804,E2 -9976.804} C_VEL
LIN {X 0,Y 426.462,Z 494.044,A -85,B 0,C 180,E1 -9977.871,E2 -9977.871} C_VEL
LIN {X 0,Y 425.779,Z 503.69,A -85,B 0,C 180,E1 -9979.298,E2 -9979.298} C_VEL
LIN {X 0,Y 425.245,Z 511.384,A -85,B 0,C 180,E1 -9980.727,E2 -9980.727} C_VEL
LIN {X 0,Y 424.683,Z 518.446,A -85,B 0,C 180,E1 -9982.392,E2 -9982.392} C_VEL
LIN {X 0,Y 424.573,Z 522.544,A -85,B 0,C 180,E1 -9983.621,E2 -9983.621} C_VEL
LIN {X 0,Y 424.285,Z 526.746,A -85,B 0,C 180,E1 -9985.249,E2 -9985.249} C_VEL
LIN {X 0,Y 424.228,Z 529.593,A -85,B 0,C 180,E1 -9986.872,E2 -9986.872} C_VEL
LIN {X 0,Y 424.152,Z 531.003,A -85,B 0,C 180,E1 -9988.101,E2 -9988.101} C_VEL
LIN {X 0,Y 424.085,Z 531.852,A -85,B 0,C 180,E1 -9990,E2 -9990} C_VEL
LIN {X 0,Y 424.092,Z 531.649,A -85,B 0,C 180,E1 -9990.973,E2 -9990.973} C_VEL
LIN {X 0,Y 423.428,Z 531.215,A -85,B 0,C 180,E1 -9991.764,E2 -9991.764} C_VEL
LIN {X 0,Y 420.58,Z 530.018,A -85,B 0,C 180,E1 -9993.044,E2 -9993.044} C_VEL
LIN {X 0,Y 418.23,Z 528.562,A -85,B 0,C 180,E1 -9994.067,E2 -9994.067} C_VEL
LIN {X 0,Y 417.306,Z 527.115,A -85,B 0,C 180,E1 -9994.847,E2 -9994.847} C_VEL
LIN {X 0,Y 417.277,Z 526.549,A -85,B 0,C 180,E1 -9995.108,E2 -9995.108} C_VEL
LIN {X 0,Y 417.501,Z 522.212,A -85,B 0,C 180,E1 -9996.767,E2 -9996.767} C_VEL
LIN {X 0,Y 417.789,Z 517.201,A -85,B 0,C 180,E1 -9998.221,E2 -9998.221} C_VEL
LIN {X 0,Y 418.301,Z 510.889,A -85,B 0,C 180,E1 -9999.672,E2 -9999.672} C_VEL
LIN {X 0,Y 418.864,Z 502.989,A -85,B 0,C 180,E1 -10001.125,E2 -10001.125} C_VEL
LIN {X 0,Y 419.647,Z 493.158,A -85,B 0,C 180,E1 -10002.575,E2 -10002.575} C_VEL
LIN {X 0,Y 420.394,Z 483.787,A -85,B 0,C 180,E1 -10003.682,E2 -10003.682} C_VEL
LIN {X 0,Y 420.936,Z 474.045,A -85,B 0,C 180,E1 -10004.627,E2 -10004.627} C_VEL
LIN {X 0,Y 421.607,Z 463.2,A -85,B 0,C 180,E1 -10005.469,E2 -10005.469} C_VEL
LIN {X 0,Y 422.149,Z 450.364,A -85,B 0,C 180,E1 -10006.24,E2 -10006.24} C_VEL
LIN {X 0,Y 419.788,Z 438.262,A -85,B 0,C 180,E1 -10006.876,E2 -10006.876} C_VEL
LIN {X 0,Y 417.321,Z 427.74,A -85,B 0,C 180,E1 -10007.323,E2 -10007.323} C_VEL
LIN {X 0,Y 417.441,Z 424.334,A -85,B 0,C 180,E1 -10009.677,E2 -10009.677} C_VEL
LIN {X 0,Y 417.503,Z 420.042,A -85,B 0,C 180,E1 -10012.779,E2 -10012.779} C_VEL
LIN {X 0,Y 417.701,Z 415.772,A -85,B 0,C 180,E1 -10015.942,E2 -10015.942} C_VEL
LIN {X 0,Y 417.872,Z 411.559,A -85,B 0,C 180,E1 -10019.192,E2 -10019.192} C_VEL
LIN {X 0,Y 418.089,Z 407.303,A -85,B 0,C 180,E1 -10022.542,E2 -10022.542} C_VEL
LIN {X 0,Y 418.128,Z 404.445,A -85,B 0,C 180,E1 -10024.854,E2 -10024.854} C_VEL
LIN {X 0,Y 418.162,Z 403.399,A -85,B 0,C 180,E1 -10026.222,E2 -10026.222} C_VEL
LIN {X 0,Y 418.255,Z 403.385,A -85,B 0,C 180,E1 -10029.381,E2 -10029.381} C_VEL
LIN {X 0,Y 418.235,Z 403.388,A -85,B 0,C 180,E1 -10032.322,E2 -10032.322} C_VEL
LIN {X 0,Y 418.24,Z 403.388,A -85,B 0,C 180,E1 -10035.109,E2 -10035.109} C_VEL
LIN {X 0,Y 418.242,Z 403.385,A -85,B 0,C 180,E1 -10037.767,E2 -10037.767} C_VEL
LIN {X 0,Y 418.26,Z 403.388,A -85,B 0,C 180,E1 -10040.619,E2 -10040.619} C_VEL
LIN {X 0,Y 418.248,Z 403.385,A -85,B 0,C 180,E1 -10043.976,E2 -10043.976} C_VEL
LIN {X 0,Y 418.26,Z 403.384,A -85,B 0,C 180,E1 -10047.156,E2 -10047.156} C_VEL
LIN {X 0,Y 418.271,Z 403.383,A -85,B 0,C 180,E1 -10050.895,E2 -10050.895} C_VEL
LIN {X 0,Y 418.271,Z 403.384,A -85,B 0,C 180,E1 -10054.096,E2 -10054.096} C_VEL
LIN {X 0,Y 418.24,Z 403.385,A -85,B 0,C 180,E1 -10057.264,E2 -10057.264} C_VEL
LIN {X 0,Y 418.286,Z 403.383,A -85,B 0,C 180,E1 -10060.364,E2 -10060.364} C_VEL
LIN {X 0,Y 418.32,Z 403.376,A -85,B 0,C 180,E1 -10063.405,E2 -10063.405} C_VEL
LIN {X 0,Y 418.349,Z 403.371,A -85,B 0,C 180,E1 -10066.999,E2 -10066.999} C_VEL
LIN {X 0,Y 418.345,Z 403.375,A -85,B 0,C 180,E1 -10070.329,E2 -10070.329} C_VEL
LIN {X 0,Y 418.497,Z 403.354,A -85,B 0,C 180,E1 -10073.249,E2 -10073.249} C_VEL
LIN {X 0,Y 418.341,Z 403.374,A -85,B 0,C 180,E1 -10075.181,E2 -10075.181} C_VEL
LIN {X 0,Y 418.545,Z 403.352,A -85,B 0,C 180,E1 -10078.075,E2 -10078.075} C_VEL
LIN {X 0,Y 418.674,Z 403.335,A -85,B 0,C 180,E1 -10080,E2 -10080} C_VEL
LIN {X 0,Y 418.504,Z 403.352,A -85,B 0,C 180,E1 -10082.888,E2 -10082.888} C_VEL
LIN {X 0,Y 418.497,Z 403.354,A -85,B 0,C 180,E1 -10086.751,E2 -10086.751} C_VEL
LIN {X 0,Y 418.363,Z 403.374,A -85,B 0,C 180,E1 -10089.671,E2 -10089.671} C_VEL
LIN {X 0,Y 418.358,Z 403.372,A -85,B 0,C 180,E1 -10093.006,E2 -10093.006} C_VEL
LIN {X 0,Y 418.316,Z 403.375,A -85,B 0,C 180,E1 -10096.736,E2 -10096.736} C_VEL
LIN {X 0,Y 418.274,Z 403.384,A -85,B 0,C 180,E1 -10099.79,E2 -10099.79} C_VEL
LIN {X 0,Y 418.24,Z 403.387,A -85,B 0,C 180,E1 -10102.736,E2 -10102.736} C_VEL
LIN {X 0,Y 418.271,Z 403.382,A -85,B 0,C 180,E1 -10105.904,E2 -10105.904} C_VEL
LIN {X 0,Y 418.267,Z 403.387,A -85,B 0,C 180,E1 -10109.162,E2 -10109.162} C_VEL
LIN {X 0,Y 418.26,Z 403.386,A -85,B 0,C 180,E1 -10112.844,E2 -10112.844} C_VEL
LIN {X 0,Y 418.251,Z 403.384,A -85,B 0,C 180,E1 -10116.239,E2 -10116.239} C_VEL
LIN {X 0,Y 418.255,Z 403.384,A -85,B 0,C 180,E1 -10119.682,E2 -10119.682} C_VEL
LIN {X 0,Y 418.232,Z 403.386,A -85,B 0,C 180,E1 -10122.321,E2 -10122.321} C_VEL
LIN {X 0,Y 418.242,Z 403.388,A -85,B 0,C 180,E1 -10125.109,E2 -10125.109} C_VEL
LIN {X 0,Y 418.245,Z 403.391,A -85,B 0,C 180,E1 -10127.767,E2 -10127.767} C_VEL
LIN {X 0,Y 418.287,Z 403.581,A -85,B 0,C 180,E1 -10129.427,E2 -10129.427} C_VEL
LIN {X 0,Y 419.064,Z 407.96,A -85,B 0,C 180,E1 -10132.02,E2 -10132.02} C_VEL
LIN {X 0,Y 419.506,Z 412.706,A -85,B 0,C 180,E1 -10134.692,E2 -10134.692} C_VEL
LIN {X 0,Y 419.085,Z 419.23,A -85,B 0,C 180,E1 -10138.112,E2 -10138.112} C_VEL
LIN {X 0,Y 418.663,Z 425.798,A -85,B 0,C 180,E1 -10141.417,E2 -10141.417} C_VEL
LIN {X 0,Y 418.212,Z 433.482,A -85,B 0,C 180,E1 -10145.158,E2 -10145.158} C_VEL
LIN {X 0,Y 417.898,Z 440,A -85,B 0,C 180,E1 -10148.285,E2 -10148.285} C_VEL
LIN {X 0,Y 417.595,Z 446.463,A -85,B 0,C 180,E1 -10151.351,E2 -10151.351} C_VEL
LIN {X 0,Y 417.51,Z 449.433,A -85,B 0,C 180,E1 -10152.725,E2 -10152.725} C_VEL
LIN {X 0,Y 419.898,Z 462.706,A -85,B 0,C 180,E1 -10153.224,E2 -10153.224} C_VEL
LIN {X 0,Y 421.678,Z 475.958,A -85,B 0,C 180,E1 -10153.914,E2 -10153.914} C_VEL
LIN {X 0,Y 421.135,Z 487.672,A -85,B 0,C 180,E1 -10154.637,E2 -10154.637} C_VEL
LIN {X 0,Y 420.347,Z 499.554,A -85,B 0,C 180,E1 -10155.589,E2 -10155.589} C_VEL
LIN {X 0,Y 419.599,Z 510.325,A -85,B 0,C 180,E1 -10156.685,E2 -10156.685} C_VEL
LIN {X 0,Y 418.95,Z 519.938,A -85,B 0,C 180,E1 -10157.896,E2 -10157.896} C_VEL
LIN {X 0,Y 418.308,Z 527.816,A -85,B 0,C 180,E1 -10159.105,E2 -10159.105} C_VEL
LIN {X 0,Y 417.795,Z 535.513,A -85,B 0,C 180,E1 -10160.56,E2 -10160.56} C_VEL
LIN {X 0,Y 417.385,Z 542.612,A -85,B 0,C 180,E1 -10162.258,E2 -10162.258} C_VEL
LIN {X 0,Y 417.146,Z 547.397,A -85,B 0,C 180,E1 -10163.734,E2 -10163.734} C_VEL
LIN {X 0,Y 417.112,Z 550.947,A -85,B 0,C 180,E1 -10165.167,E2 -10165.167} C_VEL
LIN {X 0,Y 417.016,Z 552.807,A -85,B 0,C 180,E1 -10166.135,E2 -10166.135} C_VEL
LIN {X 0,Y 417.029,Z 554.205,A -85,B 0,C 180,E1 -10167.102,E2 -10167.102} C_VEL
LIN {X 0,Y 417.056,Z 555.203,A -85,B 0,C 180,E1 -10168.068,E2 -10168.068} C_VEL
LIN {X 0,Y 417.004,Z 556.026,A -85,B 0,C 180,E1 -10170,E2 -10170} C_VEL
LIN {X 0,Y 417.056,Z 555.202,A -85,B 0,C 180,E1 -10171.931,E2 -10171.931} C_VEL
LIN {X 0,Y 417.029,Z 554.204,A -85,B 0,C 180,E1 -10172.898,E2 -10172.898} C_VEL
LIN {X 0,Y 417.016,Z 552.806,A -85,B 0,C 180,E1 -10173.865,E2 -10173.865} C_VEL
LIN {X 0,Y 417.129,Z 549.868,A -85,B 0,C 180,E1 -10175.317,E2 -10175.317} C_VEL
LIN {X 0,Y 417.235,Z 545.89,A -85,B 0,C 180,E1 -10176.771,E2 -10176.771} C_VEL
LIN {X 0,Y 417.544,Z 539.776,A -85,B 0,C 180,E1 -10178.469,E2 -10178.469} C_VEL
LIN {X 0,Y 417.942,Z 533.096,A -85,B 0,C 180,E1 -10179.925,E2 -10179.925} C_VEL
LIN {X 0,Y 418.532,Z 524.81,A -85,B 0,C 180,E1 -10181.379,E2 -10181.379} C_VEL
LIN {X 0,Y 419.218,Z 516.32,A -85,B 0,C 180,E1 -10182.588,E2 -10182.588} C_VEL
LIN {X 0,Y 419.928,Z 506.546,A -85,B 0,C 180,E1 -10183.722,E2 -10183.722} C_VEL
LIN {X 0,Y 420.5,Z 496.876,A -85,B 0,C 180,E1 -10184.643,E2 -10184.643} C_VEL
LIN {X 0,Y 421.233,Z 485.84,A -85,B 0,C 180,E1 -10185.483,E2 -10185.483} C_VEL
LIN {X 0,Y 421.649,Z 475.866,A -85,B 0,C 180,E1 -10186.087,E2 -10186.087} C_VEL
LIN {X 0,Y 419.893,Z 462.572,A -85,B 0,C 180,E1 -10186.776,E2 -10186.776} C_VEL
LIN {X 0,Y 417.532,Z 449.303,A -85,B 0,C 180,E1 -10187.295,E2 -10187.295} C_VEL
LIN {X 0,Y 417.817,Z 442.154,A -85,B 0,C 180,E1 -10190.685,E2 -10190.685} C_VEL
LIN {X 0,Y 418.059,Z 435.636,A -85,B 0,C 180,E1 -10193.795,E2 -10193.795} C_VEL
LIN {X 0,Y 418.418,Z 428.8,A -85,B 0,C 180,E1 -10197.099,E2 -10197.099} C_VEL
LIN {X 0,Y 418.877,Z 422.474,A -85,B 0,C 180,E1 -10200.222,E2 -10200.222} C_VEL
LIN {X 0,Y 419.295,Z 415.938,A -85,B 0,C 180,E1 -10203.582,E2 -10203.582} C_VEL
LIN {X 0,Y 419.441,Z 411.594,A -85,B 0,C 180,E1 -10205.905,E2 -10205.905} C_VEL
LIN {X 0,Y 418.987,Z 407.265,A -85,B 0,C 180,E1 -10208.362,E2 -10208.362} C_VEL
LIN {X 0,Y 418.252,Z 403.388,A -85,B 0,C 180,E1 -10210.794,E2 -10210.794} C_VEL
LIN {X 0,Y 418.218,Z 403.395,A -85,B 0,C 180,E1 -10213.73,E2 -10213.73} C_VEL
LIN {X 0,Y 418.21,Z 403.39,A -85,B 0,C 180,E1 -10216.449,E2 -10216.449} C_VEL
LIN {X 0,Y 418.225,Z 403.391,A -85,B 0,C 180,E1 -10219.13,E2 -10219.13} C_VEL
LIN {X 0,Y 418.236,Z 403.386,A -85,B 0,C 180,E1 -10222.165,E2 -10222.165} C_VEL
LIN {X 0,Y 418.267,Z 403.384,A -85,B 0,C 180,E1 -10225.42,E2 -10225.42} C_VEL
LIN {X 0,Y 418.213,Z 403.391,A -85,B 0,C 180,E1 -10228.604,E2 -10228.604} C_VEL
LIN {X 0,Y 418.293,Z 403.378,A -85,B 0,C 180,E1 -10231.937,E2 -10231.937} C_VEL
LIN {X 0,Y 418.291,Z 403.381,A -85,B 0,C 180,E1 -10235.163,E2 -10235.163} C_VEL
LIN {X 0,Y 418.236,Z 403.389,A -85,B 0,C 180,E1 -10238.304,E2 -10238.304} C_VEL
LIN {X 0,Y 418.286,Z 403.38,A -85,B 0,C 180,E1 -10241.383,E2 -10241.383} C_VEL
LIN {X 0,Y 418.305,Z 403.381,A -85,B 0,C 180,E1 -10244.406,E2 -10244.406} C_VEL
LIN {X 0,Y 418.372,Z 403.368,A -85,B 0,C 180,E1 -10247.386,E2 -10247.386} C_VEL
LIN {X 0,Y 418.361,Z 403.374,A -85,B 0,C 180,E1 -10250.329,E2 -10250.329} C_VEL
LIN {X 0,Y 418.496,Z 403.354,A -85,B 0,C 180,E1 -10253.249,E2 -10253.249} C_VEL
LIN {X 0,Y 418.34,Z 403.373,A -85,B 0,C 180,E1 -10255.182,E2 -10255.182} C_VEL
LIN {X 0,Y 418.544,Z 403.351,A -85,B 0,C 180,E1 -10258.076,E2 -10258.076} C_VEL
LIN {X 0,Y 418.675,Z 403.335,A -85,B 0,C 180,E1 -10260,E2 -10260} C_VEL
LIN {X 0,Y 418.502,Z 403.353,A -85,B 0,C 180,E1 -10262.888,E2 -10262.888} C_VEL
LIN {X 0,Y 418.496,Z 403.354,A -85,B 0,C 180,E1 -10266.751,E2 -10266.751} C_VEL
LIN {X 0,Y 418.362,Z 403.372,A -85,B 0,C 180,E1 -10269.671,E2 -10269.671} C_VEL
LIN {X 0,Y 418.357,Z 403.37,A -85,B 0,C 180,E1 -10273.006,E2 -10273.006} C_VEL
LIN {X 0,Y 418.314,Z 403.376,A -85,B 0,C 180,E1 -10276.735,E2 -10276.735} C_VEL
LIN {X 0,Y 418.272,Z 403.385,A -85,B 0,C 180,E1 -10279.79,E2 -10279.79} C_VEL
LIN {X 0,Y 418.239,Z 403.385,A -85,B 0,C 180,E1 -10282.736,E2 -10282.736} C_VEL
LIN {X 0,Y 418.27,Z 403.385,A -85,B 0,C 180,E1 -10285.904,E2 -10285.904} C_VEL
LIN {X 0,Y 418.266,Z 403.384,A -85,B 0,C 180,E1 -10289.162,E2 -10289.162} C_VEL
LIN {X 0,Y 418.259,Z 403.384,A -85,B 0,C 180,E1 -10292.844,E2 -10292.844} C_VEL
LIN {X 0,Y 418.251,Z 403.384,A -85,B 0,C 180,E1 -10296.239,E2 -10296.239} C_VEL
LIN {X 0,Y 418.257,Z 403.386,A -85,B 0,C 180,E1 -10299.682,E2 -10299.682} C_VEL
LIN {X 0,Y 418.231,Z 403.386,A -85,B 0,C 180,E1 -10302.321,E2 -10302.321} C_VEL
LIN {X 0,Y 418.241,Z 403.389,A -85,B 0,C 180,E1 -10305.109,E2 -10305.109} C_VEL
LIN {X 0,Y 418.244,Z 403.387,A -85,B 0,C 180,E1 -10307.767,E2 -10307.767} C_VEL
LIN {X 0,Y 418.254,Z 403.384,A -85,B 0,C 180,E1 -10310.62,E2 -10310.62} C_VEL
LIN {X 0,Y 418.165,Z 403.398,A -85,B 0,C 180,E1 -10313.968,E2 -10313.968} C_VEL
LIN {X 0,Y 418.116,Z 404.686,A -85,B 0,C 180,E1 -10315.45,E2 -10315.45} C_VEL
LIN {X 0,Y 417.991,Z 408.583,A -85,B 0,C 180,E1 -10318.585,E2 -10318.585} C_VEL
LIN {X 0,Y 417.802,Z 412.829,A -85,B 0,C 180,E1 -10321.901,E2 -10321.901} C_VEL
LIN {X 0,Y 417.648,Z 417.313,A -85,B 0,C 180,E1 -10325.325,E2 -10325.325} C_VEL
LIN {X 0,Y 417.492,Z 421.334,A -85,B 0,C 180,E1 -10328.263,E2 -10328.263} C_VEL
LIN {X 0,Y 417.392,Z 425.664,A -85,B 0,C 180,E1 -10331.342,E2 -10331.342} C_VEL
LIN {X 0,Y 417.381,Z 427.867,A -85,B 0,C 180,E1 -10332.799,E2 -10332.799} C_VEL
LIN {X 0,Y 420.444,Z 441.116,A -85,B 0,C 180,E1 -10333.36,E2 -10333.36} C_VEL
LIN {X 0,Y 422.172,Z 451.345,A -85,B 0,C 180,E1 -10333.911,E2 -10333.911} C_VEL
LIN {X 0,Y 421.593,Z 463.615,A -85,B 0,C 180,E1 -10334.655,E2 -10334.655} C_VEL
LIN {X 0,Y 420.929,Z 474.379,A -85,B 0,C 180,E1 -10335.496,E2 -10335.496} C_VEL
LIN {X 0,Y 420.252,Z 485.347,A -85,B 0,C 180,E1 -10336.583,E2 -10336.583} C_VEL
LIN {X 0,Y 419.509,Z 494.252,A -85,B 0,C 180,E1 -10337.667,E2 -10337.667} C_VEL
LIN {X 0,Y 418.817,Z 503.897,A -85,B 0,C 180,E1 -10339.118,E2 -10339.118} C_VEL
LIN {X 0,Y 418.222,Z 511.591,A -85,B 0,C 180,E1 -10340.57,E2 -10340.57} C_VEL
LIN {X 0,Y 417.654,Z 518.651,A -85,B 0,C 180,E1 -10342.264,E2 -10342.264} C_VEL
LIN {X 0,Y 417.487,Z 523.037,A -85,B 0,C 180,E1 -10343.611,E2 -10343.611} C_VEL
LIN {X 0,Y 417.223,Z 526.951,A -85,B 0,C 180,E1 -10345.169,E2 -10345.169} C_VEL
LIN {X 0,Y 417.146,Z 528.81,A -85,B 0,C 180,E1 -10346.136,E2 -10346.136} C_VEL
LIN {X 0,Y 417.158,Z 530.209,A -85,B 0,C 180,E1 -10347.103,E2 -10347.103} C_VEL
LIN {X 0,Y 417.014,Z 531.821,A -85,B 0,C 180,E1 -10349.034,E2 -10349.034} C_VEL
LIN {X 0,Y 417.004,Z 532.055,A -85,B 0,C 180,E1 -10350,E2 -10350} C_VEL
LIN {X 0,Y 417.014,Z 531.86,A -85,B 0,C 180,E1 -10350.977,E2 -10350.977} C_VEL
LIN {X 0,Y 417.154,Z 530.314,A -85,B 0,C 180,E1 -10352.897,E2 -10352.897} C_VEL
LIN {X 0,Y 417.133,Z 528.962,A -85,B 0,C 180,E1 -10353.864,E2 -10353.864} C_VEL
LIN {X 0,Y 417.277,Z 526.549,A -85,B 0,C 180,E1 -10355.108,E2 -10355.108} C_VEL
LIN {X 0,Y 416.754,Z 524.765,A -85,B 0,C 180,E1 -10355.877,E2 -10355.877} C_VEL
LIN {X 0,Y 414.072,Z 521.423,A -85,B 0,C 180,E1 -10357.11,E2 -10357.11} C_VEL
LIN {X 0,Y 411.429,Z 517.483,A -85,B 0,C 180,E1 -10358.321,E2 -10358.321} C_VEL
LIN {X 0,Y 410.982,Z 514.645,A -85,B 0,C 180,E1 -10359.047,E2 -10359.047} C_VEL
LIN {X 0,Y 411.533,Z 507.357,A -85,B 0,C 180,E1 -10360.579,E2 -10360.579} C_VEL
LIN {X 0,Y 412.278,Z 498.545,A -85,B 0,C 180,E1 -10362.054,E2 -10362.054} C_VEL
LIN {X 0,Y 413.076,Z 489.499,A -85,B 0,C 180,E1 -10363.279,E2 -10363.279} C_VEL
LIN {X 0,Y 413.713,Z 479.79,A -85,B 0,C 180,E1 -10364.356,E2 -10364.356} C_VEL
LIN {X 0,Y 414.442,Z 468.349,A -85,B 0,C 180,E1 -10365.365,E2 -10365.365} C_VEL
LIN {X 0,Y 415.165,Z 456.404,A -85,B 0,C 180,E1 -10366.184,E2 -10366.184} C_VEL
LIN {X 0,Y 415.305,Z 451.331,A -85,B 0,C 180,E1 -10366.471,E2 -10366.471} C_VEL
LIN {X 0,Y 413.057,Z 439.774,A -85,B 0,C 180,E1 -10367.109,E2 -10367.109} C_VEL
LIN {X 0,Y 410.255,Z 427.956,A -85,B 0,C 180,E1 -10367.625,E2 -10367.625} C_VEL
LIN {X 0,Y 410.36,Z 424.522,A -85,B 0,C 180,E1 -10370.031,E2 -10370.031} C_VEL
LIN {X 0,Y 410.479,Z 420.212,A -85,B 0,C 180,E1 -10373.191,E2 -10373.191} C_VEL
LIN {X 0,Y 410.605,Z 417.339,A -85,B 0,C 180,E1 -10375.335,E2 -10375.335} C_VEL
LIN {X 0,Y 410.775,Z 413.117,A -85,B 0,C 180,E1 -10378.624,E2 -10378.624} C_VEL
LIN {X 0,Y 411.002,Z 408.856,A -85,B 0,C 180,E1 -10382.012,E2 -10382.012} C_VEL
LIN {X 0,Y 411.094,Z 405.381,A -85,B 0,C 180,E1 -10384.855,E2 -10384.855} C_VEL
LIN {X 0,Y 411.077,Z 404.561,A -85,B 0,C 180,E1 -10385.541,E2 -10385.541} C_VEL
LIN {X 0,Y 411.159,Z 404.272,A -85,B 0,C 180,E1 -10386.746,E2 -10386.746} C_VEL
LIN {X 0,Y 411.215,Z 404.26,A -85,B 0,C 180,E1 -10389.728,E2 -10389.728} C_VEL
LIN {X 0,Y 411.18,Z 404.268,A -85,B 0,C 180,E1 -10393.133,E2 -10393.133} C_VEL
LIN {X 0,Y 411.171,Z 404.266,A -85,B 0,C 180,E1 -10395.881,E2 -10395.881} C_VEL
LIN {X 0,Y 411.167,Z 404.271,A -85,B 0,C 180,E1 -10398.772,E2 -10398.772} C_VEL
LIN {X 0,Y 411.213,Z 404.26,A -85,B 0,C 180,E1 -10401.83,E2 -10401.83} C_VEL
LIN {X 0,Y 411.214,Z 404.262,A -85,B 0,C 180,E1 -10405.121,E2 -10405.121} C_VEL
LIN {X 0,Y 411.169,Z 404.268,A -85,B 0,C 180,E1 -10408.003,E2 -10408.003} C_VEL
LIN {X 0,Y 411.221,Z 404.259,A -85,B 0,C 180,E1 -10411.41,E2 -10411.41} C_VEL
LIN {X 0,Y 411.24,Z 404.257,A -85,B 0,C 180,E1 -10413.619,E2 -10413.619} C_VEL
LIN {X 0,Y 411.205,Z 404.263,A -85,B 0,C 180,E1 -10416.852,E2 -10416.852} C_VEL
LIN {X 0,Y 411.218,Z 404.264,A -85,B 0,C 180,E1 -10420.05,E2 -10420.05} C_VEL
LIN {X 0,Y 411.266,Z 404.254,A -85,B 0,C 180,E1 -10423.131,E2 -10423.131} C_VEL
LIN {X 0,Y 411.309,Z 404.248,A -85,B 0,C 180,E1 -10426.896,E2 -10426.896} C_VEL
LIN {X 0,Y 411.297,Z 404.254,A -85,B 0,C 180,E1 -10430.161,E2 -10430.161} C_VEL
LIN {X 0,Y 411.464,Z 404.23,A -85,B 0,C 180,E1 -10433.133,E2 -10433.133} C_VEL
LIN {X 0,Y 411.312,Z 404.249,A -85,B 0,C 180,E1 -10435.099,E2 -10435.099} C_VEL
LIN {X 0,Y 411.514,Z 404.228,A -85,B 0,C 180,E1 -10438.043,E2 -10438.043} C_VEL
LIN {X 0,Y 411.643,Z 404.211,A -85,B 0,C 180,E1 -10440,E2 -10440} C_VEL
LIN {X 0,Y 411.461,Z 404.229,A -85,B 0,C 180,E1 -10442.937,E2 -10442.937} C_VEL
LIN {X 0,Y 411.464,Z 404.23,A -85,B 0,C 180,E1 -10446.867,E2 -10446.867} C_VEL
LIN {X 0,Y 411.311,Z 404.253,A -85,B 0,C 180,E1 -10449.838,E2 -10449.838} C_VEL
LIN {X 0,Y 411.317,Z 404.249,A -85,B 0,C 180,E1 -10453.109,E2 -10453.109} C_VEL
LIN {X 0,Y 411.26,Z 404.255,A -85,B 0,C 180,E1 -10456.889,E2 -10456.889} C_VEL
LIN {X 0,Y 411.233,Z 404.259,A -85,B 0,C 180,E1 -10459.987,E2 -10459.987} C_VEL
LIN {X 0,Y 411.205,Z 404.265,A -85,B 0,C 180,E1 -10463.147,E2 -10463.147} C_VEL
LIN {X 0,Y 411.239,Z 404.257,A -85,B 0,C 180,E1 -10466.381,E2 -10466.381} C_VEL
LIN {X 0,Y 411.203,Z 404.263,A -85,B 0,C 180,E1 -10469.713,E2 -10469.713} C_VEL
LIN {X 0,Y 411.209,Z 404.265,A -85,B 0,C 180,E1 -10473.156,E2 -10473.156} C_VEL
LIN {X 0,Y 411.198,Z 404.264,A -85,B 0,C 180,E1 -10476.553,E2 -10476.553} C_VEL
LIN {X 0,Y 411.218,Z 404.26,A -85,B 0,C 180,E1 -10479.728,E2 -10479.728} C_VEL
LIN {X 0,Y 411.175,Z 404.268,A -85,B 0,C 180,E1 -10483.133,E2 -10483.133} C_VEL
LIN {X 0,Y 411.175,Z 404.267,A -85,B 0,C 180,E1 -10485.88,E2 -10485.88} C_VEL
LIN {X 0,Y 411.236,Z 404.403,A -85,B 0,C 180,E1 -10489.138,E2 -10489.138} C_VEL
LIN {X 0,Y 412.1,Z 409.349,A -85,B 0,C 180,E1 -10492.124,E2 -10492.124} C_VEL
